DATA_BLOCK "BR04_TR07"	// DB 240
VERSION : 0.1
  STRUCT
   Front : STRUCT
    Hook : ARRAY  [1 .. 10 ] OF UDT 102;
   END_STRUCT ;
   Rear : STRUCT
    Hook : ARRAY  [1 .. 10 ] OF UDT 102;
   END_STRUCT ;
  END_STRUCT ;	
BEGIN
   Front.Hook[1].HookOver := L#6716;
   Front.Hook[1].HookUnderOffset := L#115;
   Front.Hook[1].TelPos_1.TelPos := L#3;
   Front.Hook[2].HookOver := L#5745;
   Front.Hook[2].HookUnderOffset := L#115;
   Front.Hook[2].TelPos_1.TelPos := L#3;
   Front.Hook[3].HookOver := L#4775;
   Front.Hook[3].HookUnderOffset := L#115;
   Front.Hook[3].TelPos_1.TelPos := L#3;
   Front.Hook[4].HookOver := L#3805;
   Front.Hook[4].HookUnderOffset := L#115;
   Front.Hook[4].TelPos_1.TelPos := L#3;
   Front.Hook[5].HookOver := L#2835;
   Front.Hook[5].HookUnderOffset := L#115;
   Front.Hook[5].TelPos_1.TelPos := L#3;
   Front.Hook[6].HookOver := L#1865;
   Front.Hook[6].HookUnderOffset := L#115;
   Front.Hook[6].TelPos_1.TelPos := L#3;
   Rear.Hook[1].HookOver := L#6716;
   Rear.Hook[1].HookUnderOffset := L#115;
   Rear.Hook[1].TelPos_1.TelPos := L#4;
   Rear.Hook[2].HookOver := L#5745;
   Rear.Hook[2].HookUnderOffset := L#115;
   Rear.Hook[2].TelPos_1.TelPos := L#4;
   Rear.Hook[3].HookOver := L#4775;
   Rear.Hook[3].HookUnderOffset := L#115;
   Rear.Hook[3].TelPos_1.TelPos := L#4;
   Rear.Hook[4].HookOver := L#3805;
   Rear.Hook[4].HookUnderOffset := L#115;
   Rear.Hook[4].TelPos_1.TelPos := L#4;
   Rear.Hook[5].HookOver := L#2835;
   Rear.Hook[5].HookUnderOffset := L#115;
   Rear.Hook[5].TelPos_1.TelPos := L#4;
   Rear.Hook[6].HookOver := L#1865;
   Rear.Hook[6].HookUnderOffset := L#115;
   Rear.Hook[6].TelPos_1.TelPos := L#4;
END_DATA_BLOCK

DATA_BLOCK "BR04_TR08"	// DB 241
VERSION : 0.1
  STRUCT
   Front : STRUCT
    Hook : ARRAY  [1 .. 10 ] OF UDT 102;
   END_STRUCT ;
   Rear : STRUCT
    Hook : ARRAY  [1 .. 10 ] OF UDT 102;
   END_STRUCT ;
  END_STRUCT ;	
BEGIN
   Front.Hook[1].HookOver := L#6716;
   Front.Hook[1].HookUnderOffset := L#115;
   Front.Hook[1].TelPos_1.TelPos := L#3;
   Front.Hook[2].HookOver := L#5745;
   Front.Hook[2].HookUnderOffset := L#115;
   Front.Hook[2].TelPos_1.TelPos := L#3;
   Front.Hook[3].HookOver := L#4775;
   Front.Hook[3].HookUnderOffset := L#115;
   Front.Hook[3].TelPos_1.TelPos := L#3;
   Front.Hook[4].HookOver := L#3805;
   Front.Hook[4].HookUnderOffset := L#115;
   Front.Hook[4].TelPos_1.TelPos := L#3;
   Front.Hook[5].HookOver := L#2835;
   Front.Hook[5].HookUnderOffset := L#115;
   Front.Hook[5].TelPos_1.TelPos := L#3;
   Front.Hook[6].HookOver := L#1865;
   Front.Hook[6].HookUnderOffset := L#115;
   Front.Hook[6].TelPos_1.TelPos := L#3;
   Rear.Hook[1].HookOver := L#6716;
   Rear.Hook[1].HookUnderOffset := L#115;
   Rear.Hook[1].TelPos_1.TelPos := L#4;
   Rear.Hook[2].HookOver := L#5745;
   Rear.Hook[2].HookUnderOffset := L#115;
   Rear.Hook[2].TelPos_1.TelPos := L#4;
   Rear.Hook[3].HookOver := L#4775;
   Rear.Hook[3].HookUnderOffset := L#115;
   Rear.Hook[3].TelPos_1.TelPos := L#4;
   Rear.Hook[4].HookOver := L#3805;
   Rear.Hook[4].HookUnderOffset := L#115;
   Rear.Hook[4].TelPos_1.TelPos := L#4;
   Rear.Hook[5].HookOver := L#2835;
   Rear.Hook[5].HookUnderOffset := L#115;
   Rear.Hook[5].TelPos_1.TelPos := L#4;
   Rear.Hook[6].HookOver := L#1865;
   Rear.Hook[6].HookUnderOffset := L#115;
   Rear.Hook[6].TelPos_1.TelPos := L#4;
END_DATA_BLOCK

DATA_BLOCK "BR04_TR09"	// DB 242
VERSION : 0.1
  STRUCT
   Front : STRUCT
    Hook : ARRAY  [1 .. 10 ] OF UDT 102;
   END_STRUCT ;
   Rear : STRUCT
    Hook : ARRAY  [1 .. 10 ] OF UDT 102;
   END_STRUCT ;
  END_STRUCT ;	
BEGIN
   Front.Hook[1].HookOver := L#6716;
   Front.Hook[1].HookUnderOffset := L#115;
   Front.Hook[1].TelPos_1.TelPos := L#3;
   Front.Hook[2].HookOver := L#5745;
   Front.Hook[2].HookUnderOffset := L#115;
   Front.Hook[2].TelPos_1.TelPos := L#3;
   Front.Hook[3].HookOver := L#4775;
   Front.Hook[3].HookUnderOffset := L#115;
   Front.Hook[3].TelPos_1.TelPos := L#3;
   Front.Hook[4].HookOver := L#3805;
   Front.Hook[4].HookUnderOffset := L#115;
   Front.Hook[4].TelPos_1.TelPos := L#3;
   Front.Hook[5].HookOver := L#2835;
   Front.Hook[5].HookUnderOffset := L#115;
   Front.Hook[5].TelPos_1.TelPos := L#3;
   Front.Hook[6].HookOver := L#1865;
   Front.Hook[6].HookUnderOffset := L#115;
   Front.Hook[6].TelPos_1.TelPos := L#3;
   Rear.Hook[1].HookOver := L#6716;
   Rear.Hook[1].HookUnderOffset := L#115;
   Rear.Hook[1].TelPos_1.TelPos := L#4;
   Rear.Hook[2].HookOver := L#5745;
   Rear.Hook[2].HookUnderOffset := L#115;
   Rear.Hook[2].TelPos_1.TelPos := L#4;
   Rear.Hook[3].HookOver := L#4775;
   Rear.Hook[3].HookUnderOffset := L#115;
   Rear.Hook[3].TelPos_1.TelPos := L#4;
   Rear.Hook[4].HookOver := L#3805;
   Rear.Hook[4].HookUnderOffset := L#115;
   Rear.Hook[4].TelPos_1.TelPos := L#4;
   Rear.Hook[5].HookOver := L#2835;
   Rear.Hook[5].HookUnderOffset := L#115;
   Rear.Hook[5].TelPos_1.TelPos := L#4;
   Rear.Hook[6].HookOver := L#1865;
   Rear.Hook[6].HookUnderOffset := L#115;
   Rear.Hook[6].TelPos_1.TelPos := L#4;
END_DATA_BLOCK

DATA_BLOCK "BR04_TR10"	// DB 243
VERSION : 0.1
  STRUCT
   Front : STRUCT
    Hook : ARRAY  [1 .. 10 ] OF UDT 102;
   END_STRUCT ;
   Rear : STRUCT
    Hook : ARRAY  [1 .. 10 ] OF UDT 102;
   END_STRUCT ;
  END_STRUCT ;	
BEGIN
   Front.Hook[1].HookOver := L#6716;
   Front.Hook[1].HookUnderOffset := L#115;
   Front.Hook[1].TelPos_1.TelPos := L#3;
   Front.Hook[2].HookOver := L#5745;
   Front.Hook[2].HookUnderOffset := L#115;
   Front.Hook[2].TelPos_1.TelPos := L#3;
   Front.Hook[3].HookOver := L#4775;
   Front.Hook[3].HookUnderOffset := L#115;
   Front.Hook[3].TelPos_1.TelPos := L#3;
   Front.Hook[4].HookOver := L#3805;
   Front.Hook[4].HookUnderOffset := L#115;
   Front.Hook[4].TelPos_1.TelPos := L#3;
   Front.Hook[5].HookOver := L#2835;
   Front.Hook[5].HookUnderOffset := L#115;
   Front.Hook[5].TelPos_1.TelPos := L#3;
   Rear.Hook[1].HookOver := L#6716;
   Rear.Hook[1].HookUnderOffset := L#115;
   Rear.Hook[1].TelPos_1.TelPos := L#4;
   Rear.Hook[2].HookOver := L#5745;
   Rear.Hook[2].HookUnderOffset := L#115;
   Rear.Hook[2].TelPos_1.TelPos := L#4;
   Rear.Hook[3].HookOver := L#4775;
   Rear.Hook[3].HookUnderOffset := L#115;
   Rear.Hook[3].TelPos_1.TelPos := L#4;
   Rear.Hook[4].HookOver := L#3805;
   Rear.Hook[4].HookUnderOffset := L#115;
   Rear.Hook[4].TelPos_1.TelPos := L#4;
   Rear.Hook[5].HookOver := L#2835;
   Rear.Hook[5].HookUnderOffset := L#115;
   Rear.Hook[5].TelPos_1.TelPos := L#4;
END_DATA_BLOCK

DATA_BLOCK "BR04_TR11"	// DB 244
VERSION : 0.1
  STRUCT
   Front : STRUCT
    Hook : ARRAY  [1 .. 10 ] OF UDT 102;
   END_STRUCT ;
   Rear : STRUCT
    Hook : ARRAY  [1 .. 10 ] OF UDT 102;
   END_STRUCT ;
  END_STRUCT ;	
BEGIN
   Front.Hook[1].HookOver := L#6716;
   Front.Hook[1].HookUnderOffset := L#115;
   Front.Hook[1].TelPos_1.TelPos := L#3;
   Front.Hook[2].HookOver := L#5745;
   Front.Hook[2].HookUnderOffset := L#115;
   Front.Hook[2].TelPos_1.TelPos := L#3;
   Front.Hook[3].HookOver := L#4775;
   Front.Hook[3].HookUnderOffset := L#115;
   Front.Hook[3].TelPos_1.TelPos := L#3;
   Front.Hook[4].HookOver := L#3805;
   Front.Hook[4].HookUnderOffset := L#115;
   Front.Hook[4].TelPos_1.TelPos := L#3;
   Front.Hook[5].HookOver := L#2835;
   Front.Hook[5].HookUnderOffset := L#115;
   Front.Hook[5].TelPos_1.TelPos := L#3;
   Front.Hook[6].HookOver := L#1865;
   Front.Hook[6].HookUnderOffset := L#115;
   Front.Hook[6].TelPos_1.TelPos := L#3;
   Rear.Hook[1].HookOver := L#6716;
   Rear.Hook[1].HookUnderOffset := L#115;
   Rear.Hook[1].TelPos_1.TelPos := L#4;
   Rear.Hook[2].HookOver := L#5745;
   Rear.Hook[2].HookUnderOffset := L#115;
   Rear.Hook[2].TelPos_1.TelPos := L#4;
   Rear.Hook[3].HookOver := L#4775;
   Rear.Hook[3].HookUnderOffset := L#115;
   Rear.Hook[3].TelPos_1.TelPos := L#4;
   Rear.Hook[4].HookOver := L#3805;
   Rear.Hook[4].HookUnderOffset := L#115;
   Rear.Hook[4].TelPos_1.TelPos := L#4;
   Rear.Hook[5].HookOver := L#2835;
   Rear.Hook[5].HookUnderOffset := L#115;
   Rear.Hook[5].TelPos_1.TelPos := L#4;
   Rear.Hook[6].HookOver := L#1865;
   Rear.Hook[6].HookUnderOffset := L#115;
   Rear.Hook[6].TelPos_1.TelPos := L#4;
END_DATA_BLOCK

DATA_BLOCK "BR05_TR01"	// DB 245
VERSION : 0.1
  STRUCT
   Front : STRUCT
    Hook : ARRAY  [1 .. 10 ] OF UDT 102;
   END_STRUCT ;
   Rear : STRUCT
    Hook : ARRAY  [1 .. 10 ] OF UDT 102;
   END_STRUCT ;
  END_STRUCT ;	
BEGIN
   Front.Hook[1].HookOver := L#6716;
   Front.Hook[1].HookUnderOffset := L#115;
   Front.Hook[1].TelPos_1.TelPos := L#3;
   Front.Hook[2].HookOver := L#5745;
   Front.Hook[2].HookUnderOffset := L#115;
   Front.Hook[2].TelPos_1.TelPos := L#3;
   Front.Hook[3].HookOver := L#4775;
   Front.Hook[3].HookUnderOffset := L#115;
   Front.Hook[3].TelPos_1.TelPos := L#3;
   Front.Hook[4].HookOver := L#3805;
   Front.Hook[4].HookUnderOffset := L#115;
   Front.Hook[4].TelPos_1.TelPos := L#3;
   Front.Hook[5].HookOver := L#2835;
   Front.Hook[5].HookUnderOffset := L#115;
   Front.Hook[5].TelPos_1.TelPos := L#3;
   Rear.Hook[1].HookOver := L#6716;
   Rear.Hook[1].HookUnderOffset := L#115;
   Rear.Hook[1].TelPos_1.TelPos := L#4;
   Rear.Hook[2].HookOver := L#5745;
   Rear.Hook[2].HookUnderOffset := L#115;
   Rear.Hook[2].TelPos_1.TelPos := L#4;
   Rear.Hook[3].HookOver := L#4775;
   Rear.Hook[3].HookUnderOffset := L#115;
   Rear.Hook[3].TelPos_1.TelPos := L#4;
   Rear.Hook[4].HookOver := L#3805;
   Rear.Hook[4].HookUnderOffset := L#115;
   Rear.Hook[4].TelPos_1.TelPos := L#4;
   Rear.Hook[5].HookOver := L#2835;
   Rear.Hook[5].HookUnderOffset := L#115;
   Rear.Hook[5].TelPos_1.TelPos := L#4;
END_DATA_BLOCK

DATA_BLOCK "BR05_TR02"	// DB 246
VERSION : 0.1
  STRUCT
   Front : STRUCT
    Hook : ARRAY  [1 .. 10 ] OF UDT 102;
   END_STRUCT ;
   Rear : STRUCT
    Hook : ARRAY  [1 .. 10 ] OF UDT 102;
   END_STRUCT ;
  END_STRUCT ;	
BEGIN
   Front.Hook[1].HookOver := L#6716;
   Front.Hook[1].HookUnderOffset := L#115;
   Front.Hook[1].TelPos_1.TelPos := L#3;
   Front.Hook[2].HookOver := L#5745;
   Front.Hook[2].HookUnderOffset := L#115;
   Front.Hook[2].TelPos_1.TelPos := L#3;
   Front.Hook[3].HookOver := L#4775;
   Front.Hook[3].HookUnderOffset := L#115;
   Front.Hook[3].TelPos_1.TelPos := L#3;
   Front.Hook[4].HookOver := L#3805;
   Front.Hook[4].HookUnderOffset := L#115;
   Front.Hook[4].TelPos_1.TelPos := L#3;
   Front.Hook[5].HookOver := L#2835;
   Front.Hook[5].HookUnderOffset := L#115;
   Front.Hook[5].TelPos_1.TelPos := L#3;
   Front.Hook[6].HookOver := L#1865;
   Front.Hook[6].HookUnderOffset := L#115;
   Front.Hook[6].TelPos_1.TelPos := L#3;
   Rear.Hook[1].HookOver := L#6716;
   Rear.Hook[1].HookUnderOffset := L#115;
   Rear.Hook[1].TelPos_1.TelPos := L#4;
   Rear.Hook[2].HookOver := L#5745;
   Rear.Hook[2].HookUnderOffset := L#115;
   Rear.Hook[2].TelPos_1.TelPos := L#4;
   Rear.Hook[3].HookOver := L#4775;
   Rear.Hook[3].HookUnderOffset := L#115;
   Rear.Hook[3].TelPos_1.TelPos := L#4;
   Rear.Hook[4].HookOver := L#3805;
   Rear.Hook[4].HookUnderOffset := L#115;
   Rear.Hook[4].TelPos_1.TelPos := L#4;
   Rear.Hook[5].HookOver := L#2835;
   Rear.Hook[5].HookUnderOffset := L#115;
   Rear.Hook[5].TelPos_1.TelPos := L#4;
   Rear.Hook[6].HookOver := L#1865;
   Rear.Hook[6].HookUnderOffset := L#115;
   Rear.Hook[6].TelPos_1.TelPos := L#4;
END_DATA_BLOCK

DATA_BLOCK "BR05_TR03"	// DB 247
VERSION : 0.1
  STRUCT
   Front : STRUCT
    Hook : ARRAY  [1 .. 10 ] OF UDT 102;
   END_STRUCT ;
   Rear : STRUCT
    Hook : ARRAY  [1 .. 10 ] OF UDT 102;
   END_STRUCT ;
  END_STRUCT ;	
BEGIN
   Front.Hook[1].HookOver := L#6716;
   Front.Hook[1].HookUnderOffset := L#115;
   Front.Hook[1].TelPos_1.TelPos := L#3;
   Front.Hook[2].HookOver := L#5745;
   Front.Hook[2].HookUnderOffset := L#115;
   Front.Hook[2].TelPos_1.TelPos := L#3;
   Front.Hook[3].HookOver := L#4775;
   Front.Hook[3].HookUnderOffset := L#115;
   Front.Hook[3].TelPos_1.TelPos := L#3;
   Front.Hook[4].HookOver := L#3805;
   Front.Hook[4].HookUnderOffset := L#115;
   Front.Hook[4].TelPos_1.TelPos := L#3;
   Front.Hook[5].HookOver := L#2835;
   Front.Hook[5].HookUnderOffset := L#115;
   Front.Hook[5].TelPos_1.TelPos := L#3;
   Front.Hook[6].HookOver := L#1865;
   Front.Hook[6].HookUnderOffset := L#115;
   Front.Hook[6].TelPos_1.TelPos := L#3;
   Rear.Hook[1].HookOver := L#6716;
   Rear.Hook[1].HookUnderOffset := L#115;
   Rear.Hook[1].TelPos_1.TelPos := L#4;
   Rear.Hook[2].HookOver := L#5745;
   Rear.Hook[2].HookUnderOffset := L#115;
   Rear.Hook[2].TelPos_1.TelPos := L#4;
   Rear.Hook[3].HookOver := L#4775;
   Rear.Hook[3].HookUnderOffset := L#115;
   Rear.Hook[3].TelPos_1.TelPos := L#4;
   Rear.Hook[4].HookOver := L#3805;
   Rear.Hook[4].HookUnderOffset := L#115;
   Rear.Hook[4].TelPos_1.TelPos := L#4;
   Rear.Hook[5].HookOver := L#2835;
   Rear.Hook[5].HookUnderOffset := L#115;
   Rear.Hook[5].TelPos_1.TelPos := L#4;
   Rear.Hook[6].HookOver := L#1865;
   Rear.Hook[6].HookUnderOffset := L#115;
   Rear.Hook[6].TelPos_1.TelPos := L#4;
END_DATA_BLOCK

DATA_BLOCK "BR05_TR04"	// DB 248
VERSION : 0.1
  STRUCT
   Front : STRUCT
    Hook : ARRAY  [1 .. 10 ] OF UDT 102;
   END_STRUCT ;
   Rear : STRUCT
    Hook : ARRAY  [1 .. 10 ] OF UDT 102;
   END_STRUCT ;
  END_STRUCT ;	
BEGIN
   Front.Hook[1].HookOver := L#6716;
   Front.Hook[1].HookUnderOffset := L#115;
   Front.Hook[1].TelPos_1.TelPos := L#3;
   Front.Hook[2].HookOver := L#5745;
   Front.Hook[2].HookUnderOffset := L#115;
   Front.Hook[2].TelPos_1.TelPos := L#3;
   Front.Hook[3].HookOver := L#4775;
   Front.Hook[3].HookUnderOffset := L#115;
   Front.Hook[3].TelPos_1.TelPos := L#3;
   Front.Hook[4].HookOver := L#3805;
   Front.Hook[4].HookUnderOffset := L#115;
   Front.Hook[4].TelPos_1.TelPos := L#3;
   Front.Hook[5].HookOver := L#2835;
   Front.Hook[5].HookUnderOffset := L#115;
   Front.Hook[5].TelPos_1.TelPos := L#3;
   Front.Hook[6].HookOver := L#1865;
   Front.Hook[6].HookUnderOffset := L#115;
   Front.Hook[6].TelPos_1.TelPos := L#3;
   Rear.Hook[1].HookOver := L#6716;
   Rear.Hook[1].HookUnderOffset := L#115;
   Rear.Hook[1].TelPos_1.TelPos := L#4;
   Rear.Hook[2].HookOver := L#5745;
   Rear.Hook[2].HookUnderOffset := L#115;
   Rear.Hook[2].TelPos_1.TelPos := L#4;
   Rear.Hook[3].HookOver := L#4775;
   Rear.Hook[3].HookUnderOffset := L#115;
   Rear.Hook[3].TelPos_1.TelPos := L#4;
   Rear.Hook[4].HookOver := L#3805;
   Rear.Hook[4].HookUnderOffset := L#115;
   Rear.Hook[4].TelPos_1.TelPos := L#4;
   Rear.Hook[5].HookOver := L#2835;
   Rear.Hook[5].HookUnderOffset := L#115;
   Rear.Hook[5].TelPos_1.TelPos := L#4;
   Rear.Hook[6].HookOver := L#1865;
   Rear.Hook[6].HookUnderOffset := L#115;
   Rear.Hook[6].TelPos_1.TelPos := L#4;
END_DATA_BLOCK

DATA_BLOCK "BR05_TR05"	// DB 249
VERSION : 0.1
  STRUCT
   Front : STRUCT
    Hook : ARRAY  [1 .. 10 ] OF UDT 102;
   END_STRUCT ;
   Rear : STRUCT
    Hook : ARRAY  [1 .. 10 ] OF UDT 102;
   END_STRUCT ;
  END_STRUCT ;	
BEGIN
   Front.Hook[1].HookOver := L#6716;
   Front.Hook[1].HookUnderOffset := L#115;
   Front.Hook[1].TelPos_1.TelPos := L#3;
   Front.Hook[2].HookOver := L#5745;
   Front.Hook[2].HookUnderOffset := L#115;
   Front.Hook[2].TelPos_1.TelPos := L#3;
   Front.Hook[3].HookOver := L#4775;
   Front.Hook[3].HookUnderOffset := L#115;
   Front.Hook[3].TelPos_1.TelPos := L#3;
   Front.Hook[4].HookOver := L#3805;
   Front.Hook[4].HookUnderOffset := L#115;
   Front.Hook[4].TelPos_1.TelPos := L#3;
   Front.Hook[5].HookOver := L#2835;
   Front.Hook[5].HookUnderOffset := L#115;
   Front.Hook[5].TelPos_1.TelPos := L#3;
   Front.Hook[6].HookOver := L#1865;
   Front.Hook[6].HookUnderOffset := L#115;
   Front.Hook[6].TelPos_1.TelPos := L#3;
   Rear.Hook[1].HookOver := L#6716;
   Rear.Hook[1].HookUnderOffset := L#115;
   Rear.Hook[1].TelPos_1.TelPos := L#4;
   Rear.Hook[2].HookOver := L#5745;
   Rear.Hook[2].HookUnderOffset := L#115;
   Rear.Hook[2].TelPos_1.TelPos := L#4;
   Rear.Hook[3].HookOver := L#4775;
   Rear.Hook[3].HookUnderOffset := L#115;
   Rear.Hook[3].TelPos_1.TelPos := L#4;
   Rear.Hook[4].HookOver := L#3805;
   Rear.Hook[4].HookUnderOffset := L#115;
   Rear.Hook[4].TelPos_1.TelPos := L#4;
   Rear.Hook[5].HookOver := L#2835;
   Rear.Hook[5].HookUnderOffset := L#115;
   Rear.Hook[5].TelPos_1.TelPos := L#4;
   Rear.Hook[6].HookOver := L#1865;
   Rear.Hook[6].HookUnderOffset := L#115;
   Rear.Hook[6].TelPos_1.TelPos := L#4;
END_DATA_BLOCK

DATA_BLOCK "BR05_TR06"	// DB 250
VERSION : 0.1
  STRUCT
   Front : STRUCT
    Hook : ARRAY  [1 .. 10 ] OF UDT 102;
   END_STRUCT ;
   Rear : STRUCT
    Hook : ARRAY  [1 .. 10 ] OF UDT 102;
   END_STRUCT ;
  END_STRUCT ;	
BEGIN
   Front.Hook[1].HookOver := L#6716;
   Front.Hook[1].HookUnderOffset := L#115;
   Front.Hook[1].TelPos_1.TelPos := L#3;
   Front.Hook[2].HookOver := L#5745;
   Front.Hook[2].HookUnderOffset := L#115;
   Front.Hook[2].TelPos_1.TelPos := L#3;
   Front.Hook[3].HookOver := L#4775;
   Front.Hook[3].HookUnderOffset := L#115;
   Front.Hook[3].TelPos_1.TelPos := L#3;
   Front.Hook[4].HookOver := L#3805;
   Front.Hook[4].HookUnderOffset := L#115;
   Front.Hook[4].TelPos_1.TelPos := L#3;
   Front.Hook[5].HookOver := L#2835;
   Front.Hook[5].HookUnderOffset := L#115;
   Front.Hook[5].TelPos_1.TelPos := L#3;
   Front.Hook[6].HookOver := L#1865;
   Front.Hook[6].HookUnderOffset := L#115;
   Front.Hook[6].TelPos_1.TelPos := L#3;
   Rear.Hook[1].HookOver := L#6716;
   Rear.Hook[1].HookUnderOffset := L#115;
   Rear.Hook[1].TelPos_1.TelPos := L#4;
   Rear.Hook[2].HookOver := L#5745;
   Rear.Hook[2].HookUnderOffset := L#115;
   Rear.Hook[2].TelPos_1.TelPos := L#4;
   Rear.Hook[3].HookOver := L#4775;
   Rear.Hook[3].HookUnderOffset := L#115;
   Rear.Hook[3].TelPos_1.TelPos := L#4;
   Rear.Hook[4].HookOver := L#3805;
   Rear.Hook[4].HookUnderOffset := L#115;
   Rear.Hook[4].TelPos_1.TelPos := L#4;
   Rear.Hook[5].HookOver := L#2835;
   Rear.Hook[5].HookUnderOffset := L#115;
   Rear.Hook[5].TelPos_1.TelPos := L#4;
   Rear.Hook[6].HookOver := L#1865;
   Rear.Hook[6].HookUnderOffset := L#115;
   Rear.Hook[6].TelPos_1.TelPos := L#4;
END_DATA_BLOCK

DATA_BLOCK "BR05_TR07"	// DB 251
VERSION : 0.1
  STRUCT
   Front : STRUCT
    Hook : ARRAY  [1 .. 10 ] OF UDT 102;
   END_STRUCT ;
   Rear : STRUCT
    Hook : ARRAY  [1 .. 10 ] OF UDT 102;
   END_STRUCT ;
  END_STRUCT ;	
BEGIN
   Front.Hook[1].HookOver := L#6716;
   Front.Hook[1].HookUnderOffset := L#115;
   Front.Hook[1].TelPos_1.TelPos := L#3;
   Front.Hook[2].HookOver := L#5745;
   Front.Hook[2].HookUnderOffset := L#115;
   Front.Hook[2].TelPos_1.TelPos := L#3;
   Front.Hook[3].HookOver := L#4775;
   Front.Hook[3].HookUnderOffset := L#115;
   Front.Hook[3].TelPos_1.TelPos := L#3;
   Front.Hook[4].HookOver := L#3805;
   Front.Hook[4].HookUnderOffset := L#115;
   Front.Hook[4].TelPos_1.TelPos := L#3;
   Front.Hook[5].HookOver := L#2835;
   Front.Hook[5].HookUnderOffset := L#115;
   Front.Hook[5].TelPos_1.TelPos := L#3;
   Front.Hook[6].HookOver := L#1865;
   Front.Hook[6].HookUnderOffset := L#115;
   Front.Hook[6].TelPos_1.TelPos := L#3;
   Rear.Hook[1].HookOver := L#6716;
   Rear.Hook[1].HookUnderOffset := L#115;
   Rear.Hook[1].TelPos_1.TelPos := L#4;
   Rear.Hook[2].HookOver := L#5745;
   Rear.Hook[2].HookUnderOffset := L#115;
   Rear.Hook[2].TelPos_1.TelPos := L#4;
   Rear.Hook[3].HookOver := L#4775;
   Rear.Hook[3].HookUnderOffset := L#115;
   Rear.Hook[3].TelPos_1.TelPos := L#4;
   Rear.Hook[4].HookOver := L#3805;
   Rear.Hook[4].HookUnderOffset := L#115;
   Rear.Hook[4].TelPos_1.TelPos := L#4;
   Rear.Hook[5].HookOver := L#2835;
   Rear.Hook[5].HookUnderOffset := L#115;
   Rear.Hook[5].TelPos_1.TelPos := L#4;
   Rear.Hook[6].HookOver := L#1865;
   Rear.Hook[6].HookUnderOffset := L#115;
   Rear.Hook[6].TelPos_1.TelPos := L#4;
END_DATA_BLOCK

DATA_BLOCK "BR05_TR08"	// DB 252
VERSION : 0.1
  STRUCT
   Front : STRUCT
    Hook : ARRAY  [1 .. 10 ] OF UDT 102;
   END_STRUCT ;
   Rear : STRUCT
    Hook : ARRAY  [1 .. 10 ] OF UDT 102;
   END_STRUCT ;
  END_STRUCT ;	
BEGIN
   Front.Hook[1].HookOver := L#6716;
   Front.Hook[1].HookUnderOffset := L#115;
   Front.Hook[1].TelPos_1.TelPos := L#3;
   Front.Hook[2].HookOver := L#5745;
   Front.Hook[2].HookUnderOffset := L#115;
   Front.Hook[2].TelPos_1.TelPos := L#3;
   Front.Hook[3].HookOver := L#4775;
   Front.Hook[3].HookUnderOffset := L#115;
   Front.Hook[3].TelPos_1.TelPos := L#3;
   Front.Hook[4].HookOver := L#3805;
   Front.Hook[4].HookUnderOffset := L#115;
   Front.Hook[4].TelPos_1.TelPos := L#3;
   Front.Hook[5].HookOver := L#2835;
   Front.Hook[5].HookUnderOffset := L#115;
   Front.Hook[5].TelPos_1.TelPos := L#3;
   Front.Hook[6].HookOver := L#1865;
   Front.Hook[6].HookUnderOffset := L#115;
   Front.Hook[6].TelPos_1.TelPos := L#3;
   Rear.Hook[1].HookOver := L#6716;
   Rear.Hook[1].HookUnderOffset := L#115;
   Rear.Hook[1].TelPos_1.TelPos := L#4;
   Rear.Hook[2].HookOver := L#5745;
   Rear.Hook[2].HookUnderOffset := L#115;
   Rear.Hook[2].TelPos_1.TelPos := L#4;
   Rear.Hook[3].HookOver := L#4775;
   Rear.Hook[3].HookUnderOffset := L#115;
   Rear.Hook[3].TelPos_1.TelPos := L#4;
   Rear.Hook[4].HookOver := L#3805;
   Rear.Hook[4].HookUnderOffset := L#115;
   Rear.Hook[4].TelPos_1.TelPos := L#4;
   Rear.Hook[5].HookOver := L#2835;
   Rear.Hook[5].HookUnderOffset := L#115;
   Rear.Hook[5].TelPos_1.TelPos := L#4;
   Rear.Hook[6].HookOver := L#1865;
   Rear.Hook[6].HookUnderOffset := L#115;
   Rear.Hook[6].TelPos_1.TelPos := L#4;
END_DATA_BLOCK

DATA_BLOCK "BR05_TR09"	// DB 253
VERSION : 0.1
  STRUCT
   Front : STRUCT
    Hook : ARRAY  [1 .. 10 ] OF UDT 102;
   END_STRUCT ;
   Rear : STRUCT
    Hook : ARRAY  [1 .. 10 ] OF UDT 102;
   END_STRUCT ;
  END_STRUCT ;	
BEGIN
   Front.Hook[1].HookOver := L#6716;
   Front.Hook[1].HookUnderOffset := L#115;
   Front.Hook[1].TelPos_1.TelPos := L#3;
   Front.Hook[2].HookOver := L#5745;
   Front.Hook[2].HookUnderOffset := L#115;
   Front.Hook[2].TelPos_1.TelPos := L#3;
   Front.Hook[3].HookOver := L#4775;
   Front.Hook[3].HookUnderOffset := L#115;
   Front.Hook[3].TelPos_1.TelPos := L#3;
   Front.Hook[4].HookOver := L#3805;
   Front.Hook[4].HookUnderOffset := L#115;
   Front.Hook[4].TelPos_1.TelPos := L#3;
   Front.Hook[5].HookOver := L#2835;
   Front.Hook[5].HookUnderOffset := L#115;
   Front.Hook[5].TelPos_1.TelPos := L#3;
   Front.Hook[6].HookOver := L#1865;
   Front.Hook[6].HookUnderOffset := L#115;
   Front.Hook[6].TelPos_1.TelPos := L#3;
   Rear.Hook[1].HookOver := L#6716;
   Rear.Hook[1].HookUnderOffset := L#115;
   Rear.Hook[1].TelPos_1.TelPos := L#4;
   Rear.Hook[2].HookOver := L#5745;
   Rear.Hook[2].HookUnderOffset := L#115;
   Rear.Hook[2].TelPos_1.TelPos := L#4;
   Rear.Hook[3].HookOver := L#4775;
   Rear.Hook[3].HookUnderOffset := L#115;
   Rear.Hook[3].TelPos_1.TelPos := L#4;
   Rear.Hook[4].HookOver := L#3805;
   Rear.Hook[4].HookUnderOffset := L#115;
   Rear.Hook[4].TelPos_1.TelPos := L#4;
   Rear.Hook[5].HookOver := L#2835;
   Rear.Hook[5].HookUnderOffset := L#115;
   Rear.Hook[5].TelPos_1.TelPos := L#4;
   Rear.Hook[6].HookOver := L#1865;
   Rear.Hook[6].HookUnderOffset := L#115;
   Rear.Hook[6].TelPos_1.TelPos := L#4;
END_DATA_BLOCK

DATA_BLOCK "BR05_TR10"	// DB 254
VERSION : 0.1
  STRUCT
   Front : STRUCT
    Hook : ARRAY  [1 .. 10 ] OF UDT 102;
   END_STRUCT ;
   Rear : STRUCT
    Hook : ARRAY  [1 .. 10 ] OF UDT 102;
   END_STRUCT ;
  END_STRUCT ;	
BEGIN
   Front.Hook[1].HookOver := L#6716;
   Front.Hook[1].HookUnderOffset := L#115;
   Front.Hook[1].TelPos_1.TelPos := L#3;
   Front.Hook[2].HookOver := L#5745;
   Front.Hook[2].HookUnderOffset := L#115;
   Front.Hook[2].TelPos_1.TelPos := L#3;
   Front.Hook[3].HookOver := L#4775;
   Front.Hook[3].HookUnderOffset := L#115;
   Front.Hook[3].TelPos_1.TelPos := L#3;
   Front.Hook[4].HookOver := L#3805;
   Front.Hook[4].HookUnderOffset := L#115;
   Front.Hook[4].TelPos_1.TelPos := L#3;
   Front.Hook[5].HookOver := L#2835;
   Front.Hook[5].HookUnderOffset := L#115;
   Front.Hook[5].TelPos_1.TelPos := L#3;
   Rear.Hook[1].HookOver := L#6716;
   Rear.Hook[1].HookUnderOffset := L#115;
   Rear.Hook[1].TelPos_1.TelPos := L#4;
   Rear.Hook[2].HookOver := L#5745;
   Rear.Hook[2].HookUnderOffset := L#115;
   Rear.Hook[2].TelPos_1.TelPos := L#4;
   Rear.Hook[3].HookOver := L#4775;
   Rear.Hook[3].HookUnderOffset := L#115;
   Rear.Hook[3].TelPos_1.TelPos := L#4;
   Rear.Hook[4].HookOver := L#3805;
   Rear.Hook[4].HookUnderOffset := L#115;
   Rear.Hook[4].TelPos_1.TelPos := L#4;
   Rear.Hook[5].HookOver := L#2835;
   Rear.Hook[5].HookUnderOffset := L#115;
   Rear.Hook[5].TelPos_1.TelPos := L#4;
END_DATA_BLOCK

DATA_BLOCK "BR05_TR11"	// DB 255
VERSION : 0.1
  STRUCT
   Front : STRUCT
    Hook : ARRAY  [1 .. 10 ] OF UDT 102;
   END_STRUCT ;
   Rear : STRUCT
    Hook : ARRAY  [1 .. 10 ] OF UDT 102;
   END_STRUCT ;
  END_STRUCT ;	
BEGIN
   Front.Hook[1].HookOver := L#6716;
   Front.Hook[1].HookUnderOffset := L#115;
   Front.Hook[1].TelPos_1.TelPos := L#3;
   Front.Hook[2].HookOver := L#5745;
   Front.Hook[2].HookUnderOffset := L#115;
   Front.Hook[2].TelPos_1.TelPos := L#3;
   Front.Hook[3].HookOver := L#4775;
   Front.Hook[3].HookUnderOffset := L#115;
   Front.Hook[3].TelPos_1.TelPos := L#3;
   Front.Hook[4].HookOver := L#3805;
   Front.Hook[4].HookUnderOffset := L#115;
   Front.Hook[4].TelPos_1.TelPos := L#3;
   Front.Hook[5].HookOver := L#2835;
   Front.Hook[5].HookUnderOffset := L#115;
   Front.Hook[5].TelPos_1.TelPos := L#3;
   Front.Hook[6].HookOver := L#1865;
   Front.Hook[6].HookUnderOffset := L#115;
   Front.Hook[6].TelPos_1.TelPos := L#3;
   Rear.Hook[1].HookOver := L#6716;
   Rear.Hook[1].HookUnderOffset := L#115;
   Rear.Hook[1].TelPos_1.TelPos := L#4;
   Rear.Hook[2].HookOver := L#5745;
   Rear.Hook[2].HookUnderOffset := L#115;
   Rear.Hook[2].TelPos_1.TelPos := L#4;
   Rear.Hook[3].HookOver := L#4775;
   Rear.Hook[3].HookUnderOffset := L#115;
   Rear.Hook[3].TelPos_1.TelPos := L#4;
   Rear.Hook[4].HookOver := L#3805;
   Rear.Hook[4].HookUnderOffset := L#115;
   Rear.Hook[4].TelPos_1.TelPos := L#4;
   Rear.Hook[5].HookOver := L#2835;
   Rear.Hook[5].HookUnderOffset := L#115;
   Rear.Hook[5].TelPos_1.TelPos := L#4;
   Rear.Hook[6].HookOver := L#1865;
   Rear.Hook[6].HookUnderOffset := L#115;
   Rear.Hook[6].TelPos_1.TelPos := L#4;
END_DATA_BLOCK

DATA_BLOCK "BR06_TR01"	// DB 256
VERSION : 0.1
  STRUCT
   Front : STRUCT
    Hook : ARRAY  [1 .. 10 ] OF UDT 102;
   END_STRUCT ;
   Rear : STRUCT
    Hook : ARRAY  [1 .. 10 ] OF UDT 102;
   END_STRUCT ;
  END_STRUCT ;	
BEGIN
   Front.Hook[1].HookOver := L#6650;
   Front.Hook[1].HookUnderOffset := L#115;
   Front.Hook[1].TelPos_1.TelPos := L#1;
   Front.Hook[2].HookOver := L#5566;
   Front.Hook[2].HookUnderOffset := L#115;
   Front.Hook[2].TelPos_1.TelPos := L#1;
   Front.Hook[3].HookOver := L#4416;
   Front.Hook[3].HookUnderOffset := L#115;
   Front.Hook[3].TelPos_1.TelPos := L#1;
   Front.Hook[4].HookOver := L#3266;
   Front.Hook[4].HookUnderOffset := L#115;
   Front.Hook[4].TelPos_1.TelPos := L#1;
   Rear.Hook[1].HookOver := L#6716;
   Rear.Hook[1].HookUnderOffset := L#115;
   Rear.Hook[1].TelPos_1.TelPos := L#2;
   Rear.Hook[2].HookOver := L#5566;
   Rear.Hook[2].HookUnderOffset := L#115;
   Rear.Hook[2].TelPos_1.TelPos := L#2;
   Rear.Hook[3].HookOver := L#4416;
   Rear.Hook[3].HookUnderOffset := L#115;
   Rear.Hook[3].TelPos_1.TelPos := L#2;
   Rear.Hook[4].HookOver := L#3266;
   Rear.Hook[4].HookUnderOffset := L#115;
   Rear.Hook[4].TelPos_1.TelPos := L#2;
END_DATA_BLOCK

DATA_BLOCK "BR06_TR02"	// DB 257
VERSION : 0.1
  STRUCT
   Front : STRUCT
    Hook : ARRAY  [1 .. 10 ] OF UDT 102;
   END_STRUCT ;
   Rear : STRUCT
    Hook : ARRAY  [1 .. 10 ] OF UDT 102;
   END_STRUCT ;
  END_STRUCT ;	
BEGIN
   Front.Hook[1].HookOver := L#6703;
   Front.Hook[1].HookUnderOffset := L#115;
   Front.Hook[1].TelPos_1.TelPos := L#1;
   Front.Hook[2].HookOver := L#5560;
   Front.Hook[2].HookUnderOffset := L#115;
   Front.Hook[2].TelPos_1.TelPos := L#1;
   Front.Hook[3].HookOver := L#4415;
   Front.Hook[3].HookUnderOffset := L#115;
   Front.Hook[3].TelPos_1.TelPos := L#1;
   Front.Hook[4].HookOver := L#3260;
   Front.Hook[4].HookUnderOffset := L#115;
   Front.Hook[4].TelPos_1.TelPos := L#1;
   Front.Hook[5].HookOver := L#2115;
   Front.Hook[5].HookUnderOffset := L#115;
   Front.Hook[5].TelPos_1.TelPos := L#1;
   Rear.Hook[1].HookOver := L#6703;
   Rear.Hook[1].HookUnderOffset := L#115;
   Rear.Hook[1].TelPos_1.TelPos := L#2;
   Rear.Hook[2].HookOver := L#5560;
   Rear.Hook[2].HookUnderOffset := L#115;
   Rear.Hook[2].TelPos_1.TelPos := L#2;
   Rear.Hook[3].HookOver := L#4415;
   Rear.Hook[3].HookUnderOffset := L#115;
   Rear.Hook[3].TelPos_1.TelPos := L#2;
   Rear.Hook[4].HookOver := L#3260;
   Rear.Hook[4].HookUnderOffset := L#115;
   Rear.Hook[4].TelPos_1.TelPos := L#2;
   Rear.Hook[5].HookOver := L#2115;
   Rear.Hook[5].HookUnderOffset := L#115;
   Rear.Hook[5].TelPos_1.TelPos := L#2;
END_DATA_BLOCK

DATA_BLOCK "BR06_TR03"	// DB 258
VERSION : 0.1
  STRUCT
   Front : STRUCT
    Hook : ARRAY  [1 .. 10 ] OF UDT 102;
   END_STRUCT ;
   Rear : STRUCT
    Hook : ARRAY  [1 .. 10 ] OF UDT 102;
   END_STRUCT ;
  END_STRUCT ;	
BEGIN
   Front.Hook[1].HookOver := L#6703;
   Front.Hook[1].HookUnderOffset := L#115;
   Front.Hook[1].TelPos_1.TelPos := L#1;
   Front.Hook[2].HookOver := L#5560;
   Front.Hook[2].HookUnderOffset := L#115;
   Front.Hook[2].TelPos_1.TelPos := L#1;
   Front.Hook[3].HookOver := L#4415;
   Front.Hook[3].HookUnderOffset := L#115;
   Front.Hook[3].TelPos_1.TelPos := L#1;
   Front.Hook[4].HookOver := L#3260;
   Front.Hook[4].HookUnderOffset := L#115;
   Front.Hook[4].TelPos_1.TelPos := L#1;
   Front.Hook[5].HookOver := L#2115;
   Front.Hook[5].HookUnderOffset := L#115;
   Front.Hook[5].TelPos_1.TelPos := L#1;
   Rear.Hook[1].HookOver := L#6703;
   Rear.Hook[1].HookUnderOffset := L#115;
   Rear.Hook[1].TelPos_1.TelPos := L#2;
   Rear.Hook[2].HookOver := L#5560;
   Rear.Hook[2].HookUnderOffset := L#115;
   Rear.Hook[2].TelPos_1.TelPos := L#2;
   Rear.Hook[3].HookOver := L#4415;
   Rear.Hook[3].HookUnderOffset := L#115;
   Rear.Hook[3].TelPos_1.TelPos := L#2;
   Rear.Hook[4].HookOver := L#3260;
   Rear.Hook[4].HookUnderOffset := L#115;
   Rear.Hook[4].TelPos_1.TelPos := L#2;
   Rear.Hook[5].HookOver := L#2115;
   Rear.Hook[5].HookUnderOffset := L#115;
   Rear.Hook[5].TelPos_1.TelPos := L#2;
END_DATA_BLOCK

DATA_BLOCK "BR06_TR04"	// DB 259
VERSION : 0.1
  STRUCT
   Front : STRUCT
    Hook : ARRAY  [1 .. 10 ] OF UDT 102;
   END_STRUCT ;
   Rear : STRUCT
    Hook : ARRAY  [1 .. 10 ] OF UDT 102;
   END_STRUCT ;
  END_STRUCT ;	
BEGIN
   Front.Hook[1].HookOver := L#6703;
   Front.Hook[1].HookUnderOffset := L#115;
   Front.Hook[1].TelPos_1.TelPos := L#1;
   Front.Hook[2].HookOver := L#5560;
   Front.Hook[2].HookUnderOffset := L#115;
   Front.Hook[2].TelPos_1.TelPos := L#1;
   Front.Hook[3].HookOver := L#4415;
   Front.Hook[3].HookUnderOffset := L#115;
   Front.Hook[3].TelPos_1.TelPos := L#1;
   Front.Hook[4].HookOver := L#3260;
   Front.Hook[4].HookUnderOffset := L#115;
   Front.Hook[4].TelPos_1.TelPos := L#1;
   Front.Hook[5].HookOver := L#2115;
   Front.Hook[5].HookUnderOffset := L#115;
   Front.Hook[5].TelPos_1.TelPos := L#1;
   Rear.Hook[1].HookOver := L#6703;
   Rear.Hook[1].HookUnderOffset := L#115;
   Rear.Hook[1].TelPos_1.TelPos := L#2;
   Rear.Hook[2].HookOver := L#5560;
   Rear.Hook[2].HookUnderOffset := L#115;
   Rear.Hook[2].TelPos_1.TelPos := L#2;
   Rear.Hook[3].HookOver := L#4415;
   Rear.Hook[3].HookUnderOffset := L#115;
   Rear.Hook[3].TelPos_1.TelPos := L#2;
   Rear.Hook[4].HookOver := L#3260;
   Rear.Hook[4].HookUnderOffset := L#115;
   Rear.Hook[4].TelPos_1.TelPos := L#2;
   Rear.Hook[5].HookOver := L#2115;
   Rear.Hook[5].HookUnderOffset := L#115;
   Rear.Hook[5].TelPos_1.TelPos := L#2;
END_DATA_BLOCK

DATA_BLOCK "BR06_TR05"	// DB 260
VERSION : 0.1
  STRUCT
   Front : STRUCT
    Hook : ARRAY  [1 .. 10 ] OF UDT 102;
   END_STRUCT ;
   Rear : STRUCT
    Hook : ARRAY  [1 .. 10 ] OF UDT 102;
   END_STRUCT ;
  END_STRUCT ;	
BEGIN
   Front.Hook[1].HookOver := L#6703;
   Front.Hook[1].HookUnderOffset := L#115;
   Front.Hook[1].TelPos_1.TelPos := L#1;
   Front.Hook[2].HookOver := L#5560;
   Front.Hook[2].HookUnderOffset := L#115;
   Front.Hook[2].TelPos_1.TelPos := L#1;
   Front.Hook[3].HookOver := L#4415;
   Front.Hook[3].HookUnderOffset := L#115;
   Front.Hook[3].TelPos_1.TelPos := L#1;
   Front.Hook[4].HookOver := L#3260;
   Front.Hook[4].HookUnderOffset := L#115;
   Front.Hook[4].TelPos_1.TelPos := L#1;
   Front.Hook[5].HookOver := L#2115;
   Front.Hook[5].HookUnderOffset := L#115;
   Front.Hook[5].TelPos_1.TelPos := L#1;
   Rear.Hook[1].HookOver := L#6703;
   Rear.Hook[1].HookUnderOffset := L#115;
   Rear.Hook[1].TelPos_1.TelPos := L#2;
   Rear.Hook[2].HookOver := L#5560;
   Rear.Hook[2].HookUnderOffset := L#115;
   Rear.Hook[2].TelPos_1.TelPos := L#2;
   Rear.Hook[3].HookOver := L#4415;
   Rear.Hook[3].HookUnderOffset := L#115;
   Rear.Hook[3].TelPos_1.TelPos := L#2;
   Rear.Hook[4].HookOver := L#3260;
   Rear.Hook[4].HookUnderOffset := L#115;
   Rear.Hook[4].TelPos_1.TelPos := L#2;
   Rear.Hook[5].HookOver := L#2115;
   Rear.Hook[5].HookUnderOffset := L#115;
   Rear.Hook[5].TelPos_1.TelPos := L#2;
END_DATA_BLOCK

DATA_BLOCK "BR06_TR06"	// DB 261
VERSION : 0.1
  STRUCT
   Front : STRUCT
    Hook : ARRAY  [1 .. 10 ] OF UDT 102;
   END_STRUCT ;
   Rear : STRUCT
    Hook : ARRAY  [1 .. 10 ] OF UDT 102;
   END_STRUCT ;
  END_STRUCT ;	
BEGIN
   Front.Hook[1].HookOver := L#6703;
   Front.Hook[1].HookUnderOffset := L#115;
   Front.Hook[1].TelPos_1.TelPos := L#1;
   Front.Hook[2].HookOver := L#5560;
   Front.Hook[2].HookUnderOffset := L#115;
   Front.Hook[2].TelPos_1.TelPos := L#1;
   Front.Hook[3].HookOver := L#4415;
   Front.Hook[3].HookUnderOffset := L#115;
   Front.Hook[3].TelPos_1.TelPos := L#1;
   Front.Hook[4].HookOver := L#3260;
   Front.Hook[4].HookUnderOffset := L#115;
   Front.Hook[4].TelPos_1.TelPos := L#1;
   Front.Hook[5].HookOver := L#2115;
   Front.Hook[5].HookUnderOffset := L#115;
   Front.Hook[5].TelPos_1.TelPos := L#1;
   Rear.Hook[1].HookOver := L#6703;
   Rear.Hook[1].HookUnderOffset := L#115;
   Rear.Hook[1].TelPos_1.TelPos := L#2;
   Rear.Hook[2].HookOver := L#5560;
   Rear.Hook[2].HookUnderOffset := L#115;
   Rear.Hook[2].TelPos_1.TelPos := L#2;
   Rear.Hook[3].HookOver := L#4415;
   Rear.Hook[3].HookUnderOffset := L#115;
   Rear.Hook[3].TelPos_1.TelPos := L#2;
   Rear.Hook[4].HookOver := L#3260;
   Rear.Hook[4].HookUnderOffset := L#115;
   Rear.Hook[4].TelPos_1.TelPos := L#2;
   Rear.Hook[5].HookOver := L#2115;
   Rear.Hook[5].HookUnderOffset := L#115;
   Rear.Hook[5].TelPos_1.TelPos := L#2;
END_DATA_BLOCK

DATA_BLOCK "BR06_TR07"	// DB 262
VERSION : 0.1
  STRUCT
   Front : STRUCT
    Hook : ARRAY  [1 .. 10 ] OF UDT 102;
   END_STRUCT ;
   Rear : STRUCT
    Hook : ARRAY  [1 .. 10 ] OF UDT 102;
   END_STRUCT ;
  END_STRUCT ;	
BEGIN
   Front.Hook[1].HookOver := L#6703;
   Front.Hook[1].HookUnderOffset := L#115;
   Front.Hook[1].TelPos_1.TelPos := L#1;
   Front.Hook[2].HookOver := L#5560;
   Front.Hook[2].HookUnderOffset := L#115;
   Front.Hook[2].TelPos_1.TelPos := L#1;
   Front.Hook[3].HookOver := L#4415;
   Front.Hook[3].HookUnderOffset := L#115;
   Front.Hook[3].TelPos_1.TelPos := L#1;
   Front.Hook[4].HookOver := L#3260;
   Front.Hook[4].HookUnderOffset := L#115;
   Front.Hook[4].TelPos_1.TelPos := L#1;
   Front.Hook[5].HookOver := L#2115;
   Front.Hook[5].HookUnderOffset := L#115;
   Front.Hook[5].TelPos_1.TelPos := L#1;
   Rear.Hook[1].HookOver := L#6703;
   Rear.Hook[1].HookUnderOffset := L#115;
   Rear.Hook[1].TelPos_1.TelPos := L#2;
   Rear.Hook[2].HookOver := L#5560;
   Rear.Hook[2].HookUnderOffset := L#115;
   Rear.Hook[2].TelPos_1.TelPos := L#2;
   Rear.Hook[3].HookOver := L#4415;
   Rear.Hook[3].HookUnderOffset := L#115;
   Rear.Hook[3].TelPos_1.TelPos := L#2;
   Rear.Hook[4].HookOver := L#3260;
   Rear.Hook[4].HookUnderOffset := L#115;
   Rear.Hook[4].TelPos_1.TelPos := L#2;
   Rear.Hook[5].HookOver := L#2115;
   Rear.Hook[5].HookUnderOffset := L#115;
   Rear.Hook[5].TelPos_1.TelPos := L#2;
END_DATA_BLOCK

DATA_BLOCK "BR06_TR08"	// DB 263
VERSION : 0.1
  STRUCT
   Front : STRUCT
    Hook : ARRAY  [1 .. 10 ] OF UDT 102;
   END_STRUCT ;
   Rear : STRUCT
    Hook : ARRAY  [1 .. 10 ] OF UDT 102;
   END_STRUCT ;
  END_STRUCT ;	
BEGIN
   Front.Hook[1].HookOver := L#6703;
   Front.Hook[1].HookUnderOffset := L#115;
   Front.Hook[1].TelPos_1.TelPos := L#1;
   Front.Hook[2].HookOver := L#5560;
   Front.Hook[2].HookUnderOffset := L#115;
   Front.Hook[2].TelPos_1.TelPos := L#1;
   Front.Hook[3].HookOver := L#4415;
   Front.Hook[3].HookUnderOffset := L#115;
   Front.Hook[3].TelPos_1.TelPos := L#1;
   Front.Hook[4].HookOver := L#3260;
   Front.Hook[4].HookUnderOffset := L#115;
   Front.Hook[4].TelPos_1.TelPos := L#1;
   Front.Hook[5].HookOver := L#2115;
   Front.Hook[5].HookUnderOffset := L#115;
   Front.Hook[5].TelPos_1.TelPos := L#1;
   Rear.Hook[1].HookOver := L#6703;
   Rear.Hook[1].HookUnderOffset := L#115;
   Rear.Hook[1].TelPos_1.TelPos := L#2;
   Rear.Hook[2].HookOver := L#5560;
   Rear.Hook[2].HookUnderOffset := L#115;
   Rear.Hook[2].TelPos_1.TelPos := L#2;
   Rear.Hook[3].HookOver := L#4415;
   Rear.Hook[3].HookUnderOffset := L#115;
   Rear.Hook[3].TelPos_1.TelPos := L#2;
   Rear.Hook[4].HookOver := L#3260;
   Rear.Hook[4].HookUnderOffset := L#115;
   Rear.Hook[4].TelPos_1.TelPos := L#2;
   Rear.Hook[5].HookOver := L#2115;
   Rear.Hook[5].HookUnderOffset := L#115;
   Rear.Hook[5].TelPos_1.TelPos := L#2;
END_DATA_BLOCK

DATA_BLOCK "BR06_TR09"	// DB 264
VERSION : 0.1
  STRUCT
   Front : STRUCT
    Hook : ARRAY  [1 .. 10 ] OF UDT 102;
   END_STRUCT ;
   Rear : STRUCT
    Hook : ARRAY  [1 .. 10 ] OF UDT 102;
   END_STRUCT ;
  END_STRUCT ;	
BEGIN
END_DATA_BLOCK

DATA_BLOCK "BR06_TR10"	// DB 265
VERSION : 0.1
  STRUCT
   Front : STRUCT
    Hook : ARRAY  [1 .. 10 ] OF UDT 102;
   END_STRUCT ;
   Rear : STRUCT
    Hook : ARRAY  [1 .. 10 ] OF UDT 102;
   END_STRUCT ;
  END_STRUCT ;	
BEGIN
   Front.Hook[1].HookOver := L#6703;
   Front.Hook[1].HookUnderOffset := L#115;
   Front.Hook[2].HookOver := L#5560;
   Front.Hook[2].HookUnderOffset := L#115;
   Front.Hook[3].HookOver := L#4415;
   Front.Hook[3].HookUnderOffset := L#115;
   Front.Hook[3].TelPos_1.TelPos := L#1;
   Front.Hook[4].HookOver := L#3260;
   Front.Hook[4].HookUnderOffset := L#115;
   Front.Hook[4].TelPos_1.TelPos := L#1;
   Rear.Hook[1].HookOver := L#6703;
   Rear.Hook[1].HookUnderOffset := L#115;
   Rear.Hook[1].TelPos_1.TelPos := L#2;
   Rear.Hook[2].HookOver := L#5560;
   Rear.Hook[2].HookUnderOffset := L#115;
   Rear.Hook[2].TelPos_1.TelPos := L#2;
   Rear.Hook[3].HookOver := L#4415;
   Rear.Hook[3].HookUnderOffset := L#115;
   Rear.Hook[3].TelPos_1.TelPos := L#2;
   Rear.Hook[4].HookOver := L#3260;
   Rear.Hook[4].HookUnderOffset := L#115;
   Rear.Hook[4].TelPos_1.TelPos := L#2;
END_DATA_BLOCK

DATA_BLOCK "BR06_TR11"	// DB 266
VERSION : 0.1
  STRUCT
   Front : STRUCT
    Hook : ARRAY  [1 .. 10 ] OF UDT 102;
   END_STRUCT ;
   Rear : STRUCT
    Hook : ARRAY  [1 .. 10 ] OF UDT 102;
   END_STRUCT ;
  END_STRUCT ;	
BEGIN
END_DATA_BLOCK

DATA_BLOCK "BR07_TR01"	// DB 267
VERSION : 0.1
  STRUCT
   Front : STRUCT
    Hook : ARRAY  [1 .. 10 ] OF UDT 102;
   END_STRUCT ;
   Rear : STRUCT
    Hook : ARRAY  [1 .. 10 ] OF UDT 102;
   END_STRUCT ;
  END_STRUCT ;	
BEGIN
   Front.Hook[1].HookOver := L#6716;
   Front.Hook[1].HookUnderOffset := L#115;
   Front.Hook[1].TelPos_1.TelPos := L#1;
   Front.Hook[2].HookOver := L#5566;
   Front.Hook[2].HookUnderOffset := L#115;
   Front.Hook[2].TelPos_1.TelPos := L#1;
   Front.Hook[3].HookOver := L#4416;
   Front.Hook[3].HookUnderOffset := L#115;
   Front.Hook[3].TelPos_1.TelPos := L#1;
   Front.Hook[4].HookOver := L#3266;
   Front.Hook[4].HookUnderOffset := L#115;
   Front.Hook[4].TelPos_1.TelPos := L#1;
   Rear.Hook[1].HookOver := L#6716;
   Rear.Hook[1].HookUnderOffset := L#115;
   Rear.Hook[1].TelPos_1.TelPos := L#2;
   Rear.Hook[2].HookOver := L#5566;
   Rear.Hook[2].HookUnderOffset := L#115;
   Rear.Hook[2].TelPos_1.TelPos := L#2;
   Rear.Hook[3].HookOver := L#4416;
   Rear.Hook[3].HookUnderOffset := L#115;
   Rear.Hook[3].TelPos_1.TelPos := L#2;
   Rear.Hook[4].HookOver := L#3266;
   Rear.Hook[4].HookUnderOffset := L#115;
   Rear.Hook[4].TelPos_1.TelPos := L#2;
END_DATA_BLOCK

DATA_BLOCK "BR07_TR02"	// DB 268
VERSION : 0.1
  STRUCT
   Front : STRUCT
    Hook : ARRAY  [1 .. 10 ] OF UDT 102;
   END_STRUCT ;
   Rear : STRUCT
    Hook : ARRAY  [1 .. 10 ] OF UDT 102;
   END_STRUCT ;
  END_STRUCT ;	
BEGIN
   Front.Hook[1].HookOver := L#6703;
   Front.Hook[1].HookUnderOffset := L#115;
   Front.Hook[1].TelPos_1.TelPos := L#1;
   Front.Hook[2].HookOver := L#5560;
   Front.Hook[2].HookUnderOffset := L#115;
   Front.Hook[2].TelPos_1.TelPos := L#1;
   Front.Hook[3].HookOver := L#4415;
   Front.Hook[3].HookUnderOffset := L#115;
   Front.Hook[3].TelPos_1.TelPos := L#1;
   Front.Hook[4].HookOver := L#3260;
   Front.Hook[4].HookUnderOffset := L#115;
   Front.Hook[4].TelPos_1.TelPos := L#1;
   Front.Hook[5].HookOver := L#2115;
   Front.Hook[5].HookUnderOffset := L#115;
   Front.Hook[5].TelPos_1.TelPos := L#1;
   Rear.Hook[1].HookOver := L#6703;
   Rear.Hook[1].HookUnderOffset := L#115;
   Rear.Hook[1].TelPos_1.TelPos := L#2;
   Rear.Hook[2].HookOver := L#5560;
   Rear.Hook[2].HookUnderOffset := L#115;
   Rear.Hook[2].TelPos_1.TelPos := L#2;
   Rear.Hook[3].HookOver := L#4415;
   Rear.Hook[3].HookUnderOffset := L#115;
   Rear.Hook[3].TelPos_1.TelPos := L#2;
   Rear.Hook[4].HookOver := L#3260;
   Rear.Hook[4].HookUnderOffset := L#115;
   Rear.Hook[4].TelPos_1.TelPos := L#2;
   Rear.Hook[5].HookOver := L#2115;
   Rear.Hook[5].HookUnderOffset := L#115;
   Rear.Hook[5].TelPos_1.TelPos := L#2;
END_DATA_BLOCK

DATA_BLOCK "BR07_TR03"	// DB 269
VERSION : 0.1
  STRUCT
   Front : STRUCT
    Hook : ARRAY  [1 .. 10 ] OF UDT 102;
   END_STRUCT ;
   Rear : STRUCT
    Hook : ARRAY  [1 .. 10 ] OF UDT 102;
   END_STRUCT ;
  END_STRUCT ;	
BEGIN
   Front.Hook[1].HookOver := L#6703;
   Front.Hook[1].HookUnderOffset := L#115;
   Front.Hook[1].TelPos_1.TelPos := L#1;
   Front.Hook[2].HookOver := L#5560;
   Front.Hook[2].HookUnderOffset := L#115;
   Front.Hook[2].TelPos_1.TelPos := L#1;
   Front.Hook[3].HookOver := L#4415;
   Front.Hook[3].HookUnderOffset := L#115;
   Front.Hook[3].TelPos_1.TelPos := L#1;
   Front.Hook[4].HookOver := L#3260;
   Front.Hook[4].HookUnderOffset := L#115;
   Front.Hook[4].TelPos_1.TelPos := L#1;
   Front.Hook[5].HookOver := L#2115;
   Front.Hook[5].HookUnderOffset := L#115;
   Front.Hook[5].TelPos_1.TelPos := L#1;
   Rear.Hook[1].HookOver := L#6703;
   Rear.Hook[1].HookUnderOffset := L#115;
   Rear.Hook[1].TelPos_1.TelPos := L#2;
   Rear.Hook[2].HookOver := L#5560;
   Rear.Hook[2].HookUnderOffset := L#115;
   Rear.Hook[2].TelPos_1.TelPos := L#2;
   Rear.Hook[3].HookOver := L#4415;
   Rear.Hook[3].HookUnderOffset := L#115;
   Rear.Hook[3].TelPos_1.TelPos := L#2;
   Rear.Hook[4].HookOver := L#3260;
   Rear.Hook[4].HookUnderOffset := L#115;
   Rear.Hook[4].TelPos_1.TelPos := L#2;
   Rear.Hook[5].HookOver := L#2115;
   Rear.Hook[5].HookUnderOffset := L#115;
   Rear.Hook[5].TelPos_1.TelPos := L#2;
END_DATA_BLOCK

DATA_BLOCK "BR07_TR04"	// DB 270
VERSION : 0.1
  STRUCT
   Front : STRUCT
    Hook : ARRAY  [1 .. 10 ] OF UDT 102;
   END_STRUCT ;
   Rear : STRUCT
    Hook : ARRAY  [1 .. 10 ] OF UDT 102;
   END_STRUCT ;
  END_STRUCT ;	
BEGIN
   Front.Hook[1].HookOver := L#6703;
   Front.Hook[1].HookUnderOffset := L#115;
   Front.Hook[1].TelPos_1.TelPos := L#1;
   Front.Hook[2].HookOver := L#5560;
   Front.Hook[2].HookUnderOffset := L#115;
   Front.Hook[2].TelPos_1.TelPos := L#1;
   Front.Hook[3].HookOver := L#4415;
   Front.Hook[3].HookUnderOffset := L#115;
   Front.Hook[3].TelPos_1.TelPos := L#1;
   Front.Hook[4].HookOver := L#3260;
   Front.Hook[4].HookUnderOffset := L#115;
   Front.Hook[4].TelPos_1.TelPos := L#1;
   Front.Hook[5].HookOver := L#2115;
   Front.Hook[5].HookUnderOffset := L#115;
   Front.Hook[5].TelPos_1.TelPos := L#1;
   Rear.Hook[1].HookOver := L#6703;
   Rear.Hook[1].HookUnderOffset := L#115;
   Rear.Hook[1].TelPos_1.TelPos := L#2;
   Rear.Hook[2].HookOver := L#5560;
   Rear.Hook[2].HookUnderOffset := L#115;
   Rear.Hook[2].TelPos_1.TelPos := L#2;
   Rear.Hook[3].HookOver := L#4415;
   Rear.Hook[3].HookUnderOffset := L#115;
   Rear.Hook[3].TelPos_1.TelPos := L#2;
   Rear.Hook[4].HookOver := L#3260;
   Rear.Hook[4].HookUnderOffset := L#115;
   Rear.Hook[4].TelPos_1.TelPos := L#2;
   Rear.Hook[5].HookOver := L#2115;
   Rear.Hook[5].HookUnderOffset := L#115;
   Rear.Hook[5].TelPos_1.TelPos := L#2;
END_DATA_BLOCK

DATA_BLOCK "BR07_TR05"	// DB 271
VERSION : 0.1
  STRUCT
   Front : STRUCT
    Hook : ARRAY  [1 .. 10 ] OF UDT 102;
   END_STRUCT ;
   Rear : STRUCT
    Hook : ARRAY  [1 .. 10 ] OF UDT 102;
   END_STRUCT ;
  END_STRUCT ;	
BEGIN
   Front.Hook[1].HookOver := L#6703;
   Front.Hook[1].HookUnderOffset := L#115;
   Front.Hook[1].TelPos_1.TelPos := L#1;
   Front.Hook[2].HookOver := L#5560;
   Front.Hook[2].HookUnderOffset := L#115;
   Front.Hook[2].TelPos_1.TelPos := L#1;
   Front.Hook[3].HookOver := L#4415;
   Front.Hook[3].HookUnderOffset := L#115;
   Front.Hook[3].TelPos_1.TelPos := L#1;
   Front.Hook[4].HookOver := L#3260;
   Front.Hook[4].HookUnderOffset := L#115;
   Front.Hook[4].TelPos_1.TelPos := L#1;
   Front.Hook[5].HookOver := L#2115;
   Front.Hook[5].HookUnderOffset := L#115;
   Front.Hook[5].TelPos_1.TelPos := L#1;
   Rear.Hook[1].HookOver := L#6703;
   Rear.Hook[1].HookUnderOffset := L#115;
   Rear.Hook[1].TelPos_1.TelPos := L#2;
   Rear.Hook[2].HookOver := L#5560;
   Rear.Hook[2].HookUnderOffset := L#115;
   Rear.Hook[2].TelPos_1.TelPos := L#2;
   Rear.Hook[3].HookOver := L#4415;
   Rear.Hook[3].HookUnderOffset := L#115;
   Rear.Hook[3].TelPos_1.TelPos := L#2;
   Rear.Hook[4].HookOver := L#3260;
   Rear.Hook[4].HookUnderOffset := L#115;
   Rear.Hook[4].TelPos_1.TelPos := L#2;
   Rear.Hook[5].HookOver := L#2115;
   Rear.Hook[5].HookUnderOffset := L#115;
   Rear.Hook[5].TelPos_1.TelPos := L#2;
END_DATA_BLOCK

DATA_BLOCK "BR07_TR06"	// DB 272
VERSION : 0.1
  STRUCT
   Front : STRUCT
    Hook : ARRAY  [1 .. 10 ] OF UDT 102;
   END_STRUCT ;
   Rear : STRUCT
    Hook : ARRAY  [1 .. 10 ] OF UDT 102;
   END_STRUCT ;
  END_STRUCT ;	
BEGIN
   Front.Hook[1].HookOver := L#6703;
   Front.Hook[1].HookUnderOffset := L#115;
   Front.Hook[1].TelPos_1.TelPos := L#1;
   Front.Hook[2].HookOver := L#5560;
   Front.Hook[2].HookUnderOffset := L#115;
   Front.Hook[2].TelPos_1.TelPos := L#1;
   Front.Hook[3].HookOver := L#4415;
   Front.Hook[3].HookUnderOffset := L#115;
   Front.Hook[3].TelPos_1.TelPos := L#1;
   Front.Hook[4].HookOver := L#3260;
   Front.Hook[4].HookUnderOffset := L#115;
   Front.Hook[4].TelPos_1.TelPos := L#1;
   Front.Hook[5].HookOver := L#2115;
   Front.Hook[5].HookUnderOffset := L#115;
   Front.Hook[5].TelPos_1.TelPos := L#1;
   Rear.Hook[1].HookOver := L#6703;
   Rear.Hook[1].HookUnderOffset := L#115;
   Rear.Hook[1].TelPos_1.TelPos := L#2;
   Rear.Hook[2].HookOver := L#5560;
   Rear.Hook[2].HookUnderOffset := L#115;
   Rear.Hook[2].TelPos_1.TelPos := L#2;
   Rear.Hook[3].HookOver := L#4415;
   Rear.Hook[3].HookUnderOffset := L#115;
   Rear.Hook[3].TelPos_1.TelPos := L#2;
   Rear.Hook[4].HookOver := L#3260;
   Rear.Hook[4].HookUnderOffset := L#115;
   Rear.Hook[4].TelPos_1.TelPos := L#2;
   Rear.Hook[5].HookOver := L#2115;
   Rear.Hook[5].HookUnderOffset := L#115;
   Rear.Hook[5].TelPos_1.TelPos := L#2;
END_DATA_BLOCK

DATA_BLOCK "BR07_TR07"	// DB 273
VERSION : 0.1
  STRUCT
   Front : STRUCT
    Hook : ARRAY  [1 .. 10 ] OF UDT 102;
   END_STRUCT ;
   Rear : STRUCT
    Hook : ARRAY  [1 .. 10 ] OF UDT 102;
   END_STRUCT ;
  END_STRUCT ;	
BEGIN
   Front.Hook[1].HookOver := L#6703;
   Front.Hook[1].HookUnderOffset := L#115;
   Front.Hook[1].TelPos_1.TelPos := L#1;
   Front.Hook[2].HookOver := L#5560;
   Front.Hook[2].HookUnderOffset := L#115;
   Front.Hook[2].TelPos_1.TelPos := L#1;
   Front.Hook[3].HookOver := L#4415;
   Front.Hook[3].HookUnderOffset := L#115;
   Front.Hook[3].TelPos_1.TelPos := L#1;
   Front.Hook[4].HookOver := L#3260;
   Front.Hook[4].HookUnderOffset := L#115;
   Front.Hook[4].TelPos_1.TelPos := L#1;
   Front.Hook[5].HookOver := L#2115;
   Front.Hook[5].HookUnderOffset := L#115;
   Front.Hook[5].TelPos_1.TelPos := L#1;
   Rear.Hook[1].HookOver := L#6703;
   Rear.Hook[1].HookUnderOffset := L#115;
   Rear.Hook[1].TelPos_1.TelPos := L#2;
   Rear.Hook[2].HookOver := L#5560;
   Rear.Hook[2].HookUnderOffset := L#115;
   Rear.Hook[2].TelPos_1.TelPos := L#2;
   Rear.Hook[3].HookOver := L#4415;
   Rear.Hook[3].HookUnderOffset := L#115;
   Rear.Hook[3].TelPos_1.TelPos := L#2;
   Rear.Hook[4].HookOver := L#3260;
   Rear.Hook[4].HookUnderOffset := L#115;
   Rear.Hook[4].TelPos_1.TelPos := L#2;
   Rear.Hook[5].HookOver := L#2115;
   Rear.Hook[5].HookUnderOffset := L#115;
   Rear.Hook[5].TelPos_1.TelPos := L#2;
END_DATA_BLOCK

DATA_BLOCK "BR07_TR08"	// DB 274
VERSION : 0.1
  STRUCT
   Front : STRUCT
    Hook : ARRAY  [1 .. 10 ] OF UDT 102;
   END_STRUCT ;
   Rear : STRUCT
    Hook : ARRAY  [1 .. 10 ] OF UDT 102;
   END_STRUCT ;
  END_STRUCT ;	
BEGIN
   Front.Hook[1].HookOver := L#6703;
   Front.Hook[1].HookUnderOffset := L#115;
   Front.Hook[1].TelPos_1.TelPos := L#1;
   Front.Hook[2].HookOver := L#5560;
   Front.Hook[2].HookUnderOffset := L#115;
   Front.Hook[2].TelPos_1.TelPos := L#1;
   Front.Hook[3].HookOver := L#4415;
   Front.Hook[3].HookUnderOffset := L#115;
   Front.Hook[3].TelPos_1.TelPos := L#1;
   Front.Hook[4].HookOver := L#3260;
   Front.Hook[4].HookUnderOffset := L#115;
   Front.Hook[4].TelPos_1.TelPos := L#1;
   Front.Hook[5].HookOver := L#2115;
   Front.Hook[5].HookUnderOffset := L#115;
   Front.Hook[5].TelPos_1.TelPos := L#1;
   Rear.Hook[1].HookOver := L#6703;
   Rear.Hook[1].HookUnderOffset := L#115;
   Rear.Hook[1].TelPos_1.TelPos := L#2;
   Rear.Hook[2].HookOver := L#5560;
   Rear.Hook[2].HookUnderOffset := L#115;
   Rear.Hook[2].TelPos_1.TelPos := L#2;
   Rear.Hook[3].HookOver := L#4415;
   Rear.Hook[3].HookUnderOffset := L#115;
   Rear.Hook[3].TelPos_1.TelPos := L#2;
   Rear.Hook[4].HookOver := L#3260;
   Rear.Hook[4].HookUnderOffset := L#115;
   Rear.Hook[4].TelPos_1.TelPos := L#2;
   Rear.Hook[5].HookOver := L#2115;
   Rear.Hook[5].HookUnderOffset := L#115;
   Rear.Hook[5].TelPos_1.TelPos := L#2;
END_DATA_BLOCK

DATA_BLOCK "BR07_TR09"	// DB 275
VERSION : 0.1
  STRUCT
   Front : STRUCT
    Hook : ARRAY  [1 .. 10 ] OF UDT 102;
   END_STRUCT ;
   Rear : STRUCT
    Hook : ARRAY  [1 .. 10 ] OF UDT 102;
   END_STRUCT ;
  END_STRUCT ;	
BEGIN
END_DATA_BLOCK

DATA_BLOCK "BR07_TR10"	// DB 276
VERSION : 0.1
  STRUCT
   Front : STRUCT
    Hook : ARRAY  [1 .. 10 ] OF UDT 102;
   END_STRUCT ;
   Rear : STRUCT
    Hook : ARRAY  [1 .. 10 ] OF UDT 102;
   END_STRUCT ;
  END_STRUCT ;	
BEGIN
   Front.Hook[1].HookOver := L#6703;
   Front.Hook[1].HookUnderOffset := L#115;
   Front.Hook[2].HookOver := L#5560;
   Front.Hook[2].HookUnderOffset := L#115;
   Front.Hook[3].HookOver := L#4415;
   Front.Hook[3].HookUnderOffset := L#115;
   Front.Hook[3].TelPos_1.TelPos := L#1;
   Front.Hook[4].HookOver := L#3260;
   Front.Hook[4].HookUnderOffset := L#115;
   Front.Hook[4].TelPos_1.TelPos := L#1;
   Rear.Hook[1].HookOver := L#6703;
   Rear.Hook[1].HookUnderOffset := L#115;
   Rear.Hook[1].TelPos_1.TelPos := L#2;
   Rear.Hook[2].HookOver := L#5560;
   Rear.Hook[2].HookUnderOffset := L#115;
   Rear.Hook[2].TelPos_1.TelPos := L#2;
   Rear.Hook[3].HookOver := L#4415;
   Rear.Hook[3].HookUnderOffset := L#115;
   Rear.Hook[3].TelPos_1.TelPos := L#2;
   Rear.Hook[4].HookOver := L#3260;
   Rear.Hook[4].HookUnderOffset := L#115;
   Rear.Hook[4].TelPos_1.TelPos := L#2;
END_DATA_BLOCK

DATA_BLOCK "BR07_TR11"	// DB 277
VERSION : 0.1
  STRUCT
   Front : STRUCT
    Hook : ARRAY  [1 .. 10 ] OF UDT 102;
   END_STRUCT ;
   Rear : STRUCT
    Hook : ARRAY  [1 .. 10 ] OF UDT 102;
   END_STRUCT ;
  END_STRUCT ;	
BEGIN
END_DATA_BLOCK

DATA_BLOCK "BR08_TR01"	// DB 278
VERSION : 0.1
  STRUCT
   Front : STRUCT
    Hook : ARRAY  [1 .. 10 ] OF UDT 102;
   END_STRUCT ;
   Rear : STRUCT
    Hook : ARRAY  [1 .. 10 ] OF UDT 102;
   END_STRUCT ;
  END_STRUCT ;	
BEGIN
   Front.Hook[1].HookOver := L#6650;
   Front.Hook[1].HookUnderOffset := L#115;
   Front.Hook[1].TelPos_1.TelPos := L#1;
   Front.Hook[2].HookOver := L#5566;
   Front.Hook[2].HookUnderOffset := L#115;
   Front.Hook[2].TelPos_1.TelPos := L#1;
   Front.Hook[3].HookOver := L#4416;
   Front.Hook[3].HookUnderOffset := L#115;
   Front.Hook[3].TelPos_1.TelPos := L#1;
   Front.Hook[4].HookOver := L#3266;
   Front.Hook[4].HookUnderOffset := L#115;
   Front.Hook[4].TelPos_1.TelPos := L#1;
   Rear.Hook[1].HookOver := L#6716;
   Rear.Hook[1].HookUnderOffset := L#115;
   Rear.Hook[1].TelPos_1.TelPos := L#2;
   Rear.Hook[2].HookOver := L#5566;
   Rear.Hook[2].HookUnderOffset := L#115;
   Rear.Hook[2].TelPos_1.TelPos := L#2;
   Rear.Hook[3].HookOver := L#4416;
   Rear.Hook[3].HookUnderOffset := L#115;
   Rear.Hook[3].TelPos_1.TelPos := L#2;
   Rear.Hook[4].HookOver := L#3266;
   Rear.Hook[4].HookUnderOffset := L#115;
   Rear.Hook[4].TelPos_1.TelPos := L#2;
END_DATA_BLOCK

DATA_BLOCK "BR08_TR02"	// DB 279
VERSION : 0.1
  STRUCT
   Front : STRUCT
    Hook : ARRAY  [1 .. 10 ] OF UDT 102;
   END_STRUCT ;
   Rear : STRUCT
    Hook : ARRAY  [1 .. 10 ] OF UDT 102;
   END_STRUCT ;
  END_STRUCT ;	
BEGIN
   Front.Hook[1].HookOver := L#6703;
   Front.Hook[1].HookUnderOffset := L#115;
   Front.Hook[1].TelPos_1.TelPos := L#1;
   Front.Hook[2].HookOver := L#5560;
   Front.Hook[2].HookUnderOffset := L#115;
   Front.Hook[2].TelPos_1.TelPos := L#1;
   Front.Hook[3].HookOver := L#4415;
   Front.Hook[3].HookUnderOffset := L#115;
   Front.Hook[3].TelPos_1.TelPos := L#1;
   Front.Hook[4].HookOver := L#3260;
   Front.Hook[4].HookUnderOffset := L#115;
   Front.Hook[4].TelPos_1.TelPos := L#1;
   Front.Hook[5].HookOver := L#2115;
   Front.Hook[5].HookUnderOffset := L#115;
   Front.Hook[5].TelPos_1.TelPos := L#1;
   Rear.Hook[1].HookOver := L#6703;
   Rear.Hook[1].HookUnderOffset := L#115;
   Rear.Hook[1].TelPos_1.TelPos := L#2;
   Rear.Hook[2].HookOver := L#5560;
   Rear.Hook[2].HookUnderOffset := L#115;
   Rear.Hook[2].TelPos_1.TelPos := L#2;
   Rear.Hook[3].HookOver := L#4415;
   Rear.Hook[3].HookUnderOffset := L#115;
   Rear.Hook[3].TelPos_1.TelPos := L#2;
   Rear.Hook[4].HookOver := L#3260;
   Rear.Hook[4].HookUnderOffset := L#115;
   Rear.Hook[4].TelPos_1.TelPos := L#2;
   Rear.Hook[5].HookOver := L#2115;
   Rear.Hook[5].HookUnderOffset := L#115;
   Rear.Hook[5].TelPos_1.TelPos := L#2;
END_DATA_BLOCK

DATA_BLOCK "BR08_TR03"	// DB 280
VERSION : 0.1
  STRUCT
   Front : STRUCT
    Hook : ARRAY  [1 .. 10 ] OF UDT 102;
   END_STRUCT ;
   Rear : STRUCT
    Hook : ARRAY  [1 .. 10 ] OF UDT 102;
   END_STRUCT ;
  END_STRUCT ;	
BEGIN
   Front.Hook[1].HookOver := L#6703;
   Front.Hook[1].HookUnderOffset := L#115;
   Front.Hook[1].TelPos_1.TelPos := L#1;
   Front.Hook[2].HookOver := L#5560;
   Front.Hook[2].HookUnderOffset := L#115;
   Front.Hook[2].TelPos_1.TelPos := L#1;
   Front.Hook[3].HookOver := L#4415;
   Front.Hook[3].HookUnderOffset := L#115;
   Front.Hook[3].TelPos_1.TelPos := L#1;
   Front.Hook[4].HookOver := L#3260;
   Front.Hook[4].HookUnderOffset := L#115;
   Front.Hook[4].TelPos_1.TelPos := L#1;
   Front.Hook[5].HookOver := L#2115;
   Front.Hook[5].HookUnderOffset := L#115;
   Front.Hook[5].TelPos_1.TelPos := L#1;
   Rear.Hook[1].HookOver := L#6703;
   Rear.Hook[1].HookUnderOffset := L#115;
   Rear.Hook[1].TelPos_1.TelPos := L#2;
   Rear.Hook[2].HookOver := L#5560;
   Rear.Hook[2].HookUnderOffset := L#115;
   Rear.Hook[2].TelPos_1.TelPos := L#2;
   Rear.Hook[3].HookOver := L#4415;
   Rear.Hook[3].HookUnderOffset := L#115;
   Rear.Hook[3].TelPos_1.TelPos := L#2;
   Rear.Hook[4].HookOver := L#3260;
   Rear.Hook[4].HookUnderOffset := L#115;
   Rear.Hook[4].TelPos_1.TelPos := L#2;
   Rear.Hook[5].HookOver := L#2115;
   Rear.Hook[5].HookUnderOffset := L#115;
   Rear.Hook[5].TelPos_1.TelPos := L#2;
END_DATA_BLOCK

DATA_BLOCK "BR08_TR04"	// DB 281
VERSION : 0.1
  STRUCT
   Front : STRUCT
    Hook : ARRAY  [1 .. 10 ] OF UDT 102;
   END_STRUCT ;
   Rear : STRUCT
    Hook : ARRAY  [1 .. 10 ] OF UDT 102;
   END_STRUCT ;
  END_STRUCT ;	
BEGIN
   Front.Hook[1].HookOver := L#6703;
   Front.Hook[1].HookUnderOffset := L#115;
   Front.Hook[1].TelPos_1.TelPos := L#1;
   Front.Hook[2].HookOver := L#5560;
   Front.Hook[2].HookUnderOffset := L#115;
   Front.Hook[2].TelPos_1.TelPos := L#1;
   Front.Hook[3].HookOver := L#4415;
   Front.Hook[3].HookUnderOffset := L#115;
   Front.Hook[3].TelPos_1.TelPos := L#1;
   Front.Hook[4].HookOver := L#3260;
   Front.Hook[4].HookUnderOffset := L#115;
   Front.Hook[4].TelPos_1.TelPos := L#1;
   Front.Hook[5].HookOver := L#2115;
   Front.Hook[5].HookUnderOffset := L#115;
   Front.Hook[5].TelPos_1.TelPos := L#1;
   Rear.Hook[1].HookOver := L#6703;
   Rear.Hook[1].HookUnderOffset := L#115;
   Rear.Hook[1].TelPos_1.TelPos := L#2;
   Rear.Hook[2].HookOver := L#5560;
   Rear.Hook[2].HookUnderOffset := L#115;
   Rear.Hook[2].TelPos_1.TelPos := L#2;
   Rear.Hook[3].HookOver := L#4415;
   Rear.Hook[3].HookUnderOffset := L#115;
   Rear.Hook[3].TelPos_1.TelPos := L#2;
   Rear.Hook[4].HookOver := L#3260;
   Rear.Hook[4].HookUnderOffset := L#115;
   Rear.Hook[4].TelPos_1.TelPos := L#2;
   Rear.Hook[5].HookOver := L#2115;
   Rear.Hook[5].HookUnderOffset := L#115;
   Rear.Hook[5].TelPos_1.TelPos := L#2;
END_DATA_BLOCK

DATA_BLOCK "BR08_TR05"	// DB 282
VERSION : 0.1
  STRUCT
   Front : STRUCT
    Hook : ARRAY  [1 .. 10 ] OF UDT 102;
   END_STRUCT ;
   Rear : STRUCT
    Hook : ARRAY  [1 .. 10 ] OF UDT 102;
   END_STRUCT ;
  END_STRUCT ;	
BEGIN
   Front.Hook[1].HookOver := L#6703;
   Front.Hook[1].HookUnderOffset := L#115;
   Front.Hook[1].TelPos_1.TelPos := L#1;
   Front.Hook[2].HookOver := L#5560;
   Front.Hook[2].HookUnderOffset := L#115;
   Front.Hook[2].TelPos_1.TelPos := L#1;
   Front.Hook[3].HookOver := L#4415;
   Front.Hook[3].HookUnderOffset := L#115;
   Front.Hook[3].TelPos_1.TelPos := L#1;
   Front.Hook[4].HookOver := L#3260;
   Front.Hook[4].HookUnderOffset := L#115;
   Front.Hook[4].TelPos_1.TelPos := L#1;
   Front.Hook[5].HookOver := L#2115;
   Front.Hook[5].HookUnderOffset := L#115;
   Front.Hook[5].TelPos_1.TelPos := L#1;
   Rear.Hook[1].HookOver := L#6703;
   Rear.Hook[1].HookUnderOffset := L#115;
   Rear.Hook[1].TelPos_1.TelPos := L#2;
   Rear.Hook[2].HookOver := L#5560;
   Rear.Hook[2].HookUnderOffset := L#115;
   Rear.Hook[2].TelPos_1.TelPos := L#2;
   Rear.Hook[3].HookOver := L#4415;
   Rear.Hook[3].HookUnderOffset := L#115;
   Rear.Hook[3].TelPos_1.TelPos := L#2;
   Rear.Hook[4].HookOver := L#3260;
   Rear.Hook[4].HookUnderOffset := L#115;
   Rear.Hook[4].TelPos_1.TelPos := L#2;
   Rear.Hook[5].HookOver := L#2115;
   Rear.Hook[5].HookUnderOffset := L#115;
   Rear.Hook[5].TelPos_1.TelPos := L#2;
END_DATA_BLOCK

DATA_BLOCK "BR08_TR06"	// DB 283
VERSION : 0.1
  STRUCT
   Front : STRUCT
    Hook : ARRAY  [1 .. 10 ] OF UDT 102;
   END_STRUCT ;
   Rear : STRUCT
    Hook : ARRAY  [1 .. 10 ] OF UDT 102;
   END_STRUCT ;
  END_STRUCT ;	
BEGIN
   Front.Hook[1].HookOver := L#6703;
   Front.Hook[1].HookUnderOffset := L#115;
   Front.Hook[1].TelPos_1.TelPos := L#1;
   Front.Hook[2].HookOver := L#5560;
   Front.Hook[2].HookUnderOffset := L#115;
   Front.Hook[2].TelPos_1.TelPos := L#1;
   Front.Hook[3].HookOver := L#4415;
   Front.Hook[3].HookUnderOffset := L#115;
   Front.Hook[3].TelPos_1.TelPos := L#1;
   Front.Hook[4].HookOver := L#3260;
   Front.Hook[4].HookUnderOffset := L#115;
   Front.Hook[4].TelPos_1.TelPos := L#1;
   Front.Hook[5].HookOver := L#2115;
   Front.Hook[5].HookUnderOffset := L#115;
   Front.Hook[5].TelPos_1.TelPos := L#1;
   Rear.Hook[1].HookOver := L#6703;
   Rear.Hook[1].HookUnderOffset := L#115;
   Rear.Hook[1].TelPos_1.TelPos := L#2;
   Rear.Hook[2].HookOver := L#5560;
   Rear.Hook[2].HookUnderOffset := L#115;
   Rear.Hook[2].TelPos_1.TelPos := L#2;
   Rear.Hook[3].HookOver := L#4415;
   Rear.Hook[3].HookUnderOffset := L#115;
   Rear.Hook[3].TelPos_1.TelPos := L#2;
   Rear.Hook[4].HookOver := L#3260;
   Rear.Hook[4].HookUnderOffset := L#115;
   Rear.Hook[4].TelPos_1.TelPos := L#2;
   Rear.Hook[5].HookOver := L#2115;
   Rear.Hook[5].HookUnderOffset := L#115;
   Rear.Hook[5].TelPos_1.TelPos := L#2;
END_DATA_BLOCK

DATA_BLOCK "BR08_TR07"	// DB 284
VERSION : 0.1
  STRUCT
   Front : STRUCT
    Hook : ARRAY  [1 .. 10 ] OF UDT 102;
   END_STRUCT ;
   Rear : STRUCT
    Hook : ARRAY  [1 .. 10 ] OF UDT 102;
   END_STRUCT ;
  END_STRUCT ;	
BEGIN
   Front.Hook[1].HookOver := L#6703;
   Front.Hook[1].HookUnderOffset := L#115;
   Front.Hook[1].TelPos_1.TelPos := L#1;
   Front.Hook[2].HookOver := L#5560;
   Front.Hook[2].HookUnderOffset := L#115;
   Front.Hook[2].TelPos_1.TelPos := L#1;
   Front.Hook[3].HookOver := L#4415;
   Front.Hook[3].HookUnderOffset := L#115;
   Front.Hook[3].TelPos_1.TelPos := L#1;
   Front.Hook[4].HookOver := L#3260;
   Front.Hook[4].HookUnderOffset := L#115;
   Front.Hook[4].TelPos_1.TelPos := L#1;
   Front.Hook[5].HookOver := L#2115;
   Front.Hook[5].HookUnderOffset := L#115;
   Front.Hook[5].TelPos_1.TelPos := L#1;
   Rear.Hook[1].HookOver := L#6703;
   Rear.Hook[1].HookUnderOffset := L#115;
   Rear.Hook[1].TelPos_1.TelPos := L#2;
   Rear.Hook[2].HookOver := L#5560;
   Rear.Hook[2].HookUnderOffset := L#115;
   Rear.Hook[2].TelPos_1.TelPos := L#2;
   Rear.Hook[3].HookOver := L#4415;
   Rear.Hook[3].HookUnderOffset := L#115;
   Rear.Hook[3].TelPos_1.TelPos := L#2;
   Rear.Hook[4].HookOver := L#3260;
   Rear.Hook[4].HookUnderOffset := L#115;
   Rear.Hook[4].TelPos_1.TelPos := L#2;
   Rear.Hook[5].HookOver := L#2115;
   Rear.Hook[5].HookUnderOffset := L#115;
   Rear.Hook[5].TelPos_1.TelPos := L#2;
END_DATA_BLOCK

DATA_BLOCK "BR08_TR08"	// DB 285
VERSION : 0.1
  STRUCT
   Front : STRUCT
    Hook : ARRAY  [1 .. 10 ] OF UDT 102;
   END_STRUCT ;
   Rear : STRUCT
    Hook : ARRAY  [1 .. 10 ] OF UDT 102;
   END_STRUCT ;
  END_STRUCT ;	
BEGIN
   Front.Hook[1].HookOver := L#6703;
   Front.Hook[1].HookUnderOffset := L#115;
   Front.Hook[1].TelPos_1.TelPos := L#1;
   Front.Hook[2].HookOver := L#5560;
   Front.Hook[2].HookUnderOffset := L#115;
   Front.Hook[2].TelPos_1.TelPos := L#1;
   Front.Hook[3].HookOver := L#4415;
   Front.Hook[3].HookUnderOffset := L#115;
   Front.Hook[3].TelPos_1.TelPos := L#1;
   Front.Hook[4].HookOver := L#3260;
   Front.Hook[4].HookUnderOffset := L#115;
   Front.Hook[4].TelPos_1.TelPos := L#1;
   Front.Hook[5].HookOver := L#2115;
   Front.Hook[5].HookUnderOffset := L#115;
   Front.Hook[5].TelPos_1.TelPos := L#1;
   Rear.Hook[1].HookOver := L#6703;
   Rear.Hook[1].HookUnderOffset := L#115;
   Rear.Hook[1].TelPos_1.TelPos := L#2;
   Rear.Hook[2].HookOver := L#5560;
   Rear.Hook[2].HookUnderOffset := L#115;
   Rear.Hook[2].TelPos_1.TelPos := L#2;
   Rear.Hook[3].HookOver := L#4415;
   Rear.Hook[3].HookUnderOffset := L#115;
   Rear.Hook[3].TelPos_1.TelPos := L#2;
   Rear.Hook[4].HookOver := L#3260;
   Rear.Hook[4].HookUnderOffset := L#115;
   Rear.Hook[4].TelPos_1.TelPos := L#2;
   Rear.Hook[5].HookOver := L#2115;
   Rear.Hook[5].HookUnderOffset := L#115;
   Rear.Hook[5].TelPos_1.TelPos := L#2;
END_DATA_BLOCK

DATA_BLOCK "BR08_TR09"	// DB 286
VERSION : 0.1
  STRUCT
   Front : STRUCT
    Hook : ARRAY  [1 .. 10 ] OF UDT 102;
   END_STRUCT ;
   Rear : STRUCT
    Hook : ARRAY  [1 .. 10 ] OF UDT 102;
   END_STRUCT ;
  END_STRUCT ;	
BEGIN
END_DATA_BLOCK

DATA_BLOCK "BR08_TR10"	// DB 287
VERSION : 0.1
  STRUCT
   Front : STRUCT
    Hook : ARRAY  [1 .. 10 ] OF UDT 102;
   END_STRUCT ;
   Rear : STRUCT
    Hook : ARRAY  [1 .. 10 ] OF UDT 102;
   END_STRUCT ;
  END_STRUCT ;	
BEGIN
   Front.Hook[1].HookOver := L#6703;
   Front.Hook[1].HookUnderOffset := L#115;
   Front.Hook[2].HookOver := L#5560;
   Front.Hook[2].HookUnderOffset := L#115;
   Front.Hook[3].HookOver := L#4415;
   Front.Hook[3].HookUnderOffset := L#115;
   Front.Hook[3].TelPos_1.TelPos := L#1;
   Front.Hook[4].HookOver := L#3260;
   Front.Hook[4].HookUnderOffset := L#115;
   Front.Hook[4].TelPos_1.TelPos := L#1;
   Rear.Hook[1].HookOver := L#6703;
   Rear.Hook[1].HookUnderOffset := L#115;
   Rear.Hook[1].TelPos_1.TelPos := L#2;
   Rear.Hook[2].HookOver := L#5560;
   Rear.Hook[2].HookUnderOffset := L#115;
   Rear.Hook[2].TelPos_1.TelPos := L#2;
   Rear.Hook[3].HookOver := L#4415;
   Rear.Hook[3].HookUnderOffset := L#115;
   Rear.Hook[3].TelPos_1.TelPos := L#2;
   Rear.Hook[4].HookOver := L#3260;
   Rear.Hook[4].HookUnderOffset := L#115;
   Rear.Hook[4].TelPos_1.TelPos := L#2;
END_DATA_BLOCK

DATA_BLOCK "BR08_TR11"	// DB 288
VERSION : 0.1
  STRUCT
   Front : STRUCT
    Hook : ARRAY  [1 .. 10 ] OF UDT 102;
   END_STRUCT ;
   Rear : STRUCT
    Hook : ARRAY  [1 .. 10 ] OF UDT 102;
   END_STRUCT ;
  END_STRUCT ;	
BEGIN
END_DATA_BLOCK

DATA_BLOCK "BR09_TR01"	// DB 289
VERSION : 0.1
  STRUCT
   Front : STRUCT
    Hook : ARRAY  [1 .. 10 ] OF UDT 102;
   END_STRUCT ;
   Rear : STRUCT
    Hook : ARRAY  [1 .. 10 ] OF UDT 102;
   END_STRUCT ;
  END_STRUCT ;	
BEGIN
   Front.Hook[1].HookOver := L#6716;
   Front.Hook[1].HookUnderOffset := L#115;
   Front.Hook[1].TelPos_1.TelPos := L#1;
   Front.Hook[2].HookOver := L#5566;
   Front.Hook[2].HookUnderOffset := L#115;
   Front.Hook[2].TelPos_1.TelPos := L#1;
   Front.Hook[3].HookOver := L#4416;
   Front.Hook[3].HookUnderOffset := L#115;
   Front.Hook[3].TelPos_1.TelPos := L#1;
   Front.Hook[4].HookOver := L#3266;
   Front.Hook[4].HookUnderOffset := L#115;
   Front.Hook[4].TelPos_1.TelPos := L#1;
   Rear.Hook[1].HookOver := L#6716;
   Rear.Hook[1].HookUnderOffset := L#115;
   Rear.Hook[1].TelPos_1.TelPos := L#2;
   Rear.Hook[2].HookOver := L#5566;
   Rear.Hook[2].HookUnderOffset := L#115;
   Rear.Hook[2].TelPos_1.TelPos := L#2;
   Rear.Hook[3].HookOver := L#4416;
   Rear.Hook[3].HookUnderOffset := L#115;
   Rear.Hook[3].TelPos_1.TelPos := L#2;
   Rear.Hook[4].HookOver := L#3266;
   Rear.Hook[4].HookUnderOffset := L#115;
   Rear.Hook[4].TelPos_1.TelPos := L#2;
END_DATA_BLOCK

DATA_BLOCK "BR09_TR02"	// DB 290
VERSION : 0.1
  STRUCT
   Front : STRUCT
    Hook : ARRAY  [1 .. 10 ] OF UDT 102;
   END_STRUCT ;
   Rear : STRUCT
    Hook : ARRAY  [1 .. 10 ] OF UDT 102;
   END_STRUCT ;
  END_STRUCT ;	
BEGIN
   Front.Hook[1].HookOver := L#6703;
   Front.Hook[1].HookUnderOffset := L#115;
   Front.Hook[1].TelPos_1.TelPos := L#1;
   Front.Hook[2].HookOver := L#5560;
   Front.Hook[2].HookUnderOffset := L#115;
   Front.Hook[2].TelPos_1.TelPos := L#1;
   Front.Hook[3].HookOver := L#4415;
   Front.Hook[3].HookUnderOffset := L#115;
   Front.Hook[3].TelPos_1.TelPos := L#1;
   Front.Hook[4].HookOver := L#3260;
   Front.Hook[4].HookUnderOffset := L#115;
   Front.Hook[4].TelPos_1.TelPos := L#1;
   Front.Hook[5].HookOver := L#2115;
   Front.Hook[5].HookUnderOffset := L#115;
   Front.Hook[5].TelPos_1.TelPos := L#1;
   Rear.Hook[1].HookOver := L#6703;
   Rear.Hook[1].HookUnderOffset := L#115;
   Rear.Hook[1].TelPos_1.TelPos := L#2;
   Rear.Hook[2].HookOver := L#5560;
   Rear.Hook[2].HookUnderOffset := L#115;
   Rear.Hook[2].TelPos_1.TelPos := L#2;
   Rear.Hook[3].HookOver := L#4415;
   Rear.Hook[3].HookUnderOffset := L#115;
   Rear.Hook[3].TelPos_1.TelPos := L#2;
   Rear.Hook[4].HookOver := L#3260;
   Rear.Hook[4].HookUnderOffset := L#115;
   Rear.Hook[4].TelPos_1.TelPos := L#2;
   Rear.Hook[5].HookOver := L#2115;
   Rear.Hook[5].HookUnderOffset := L#115;
   Rear.Hook[5].TelPos_1.TelPos := L#2;
END_DATA_BLOCK

DATA_BLOCK "BR09_TR03"	// DB 291
VERSION : 0.1
  STRUCT
   Front : STRUCT
    Hook : ARRAY  [1 .. 10 ] OF UDT 102;
   END_STRUCT ;
   Rear : STRUCT
    Hook : ARRAY  [1 .. 10 ] OF UDT 102;
   END_STRUCT ;
  END_STRUCT ;	
BEGIN
   Front.Hook[1].HookOver := L#6703;
   Front.Hook[1].HookUnderOffset := L#115;
   Front.Hook[1].TelPos_1.TelPos := L#1;
   Front.Hook[2].HookOver := L#5560;
   Front.Hook[2].HookUnderOffset := L#115;
   Front.Hook[2].TelPos_1.TelPos := L#1;
   Front.Hook[3].HookOver := L#4415;
   Front.Hook[3].HookUnderOffset := L#115;
   Front.Hook[3].TelPos_1.TelPos := L#1;
   Front.Hook[4].HookOver := L#3260;
   Front.Hook[4].HookUnderOffset := L#115;
   Front.Hook[4].TelPos_1.TelPos := L#1;
   Front.Hook[5].HookOver := L#2115;
   Front.Hook[5].HookUnderOffset := L#115;
   Front.Hook[5].TelPos_1.TelPos := L#1;
   Rear.Hook[1].HookOver := L#6703;
   Rear.Hook[1].HookUnderOffset := L#115;
   Rear.Hook[1].TelPos_1.TelPos := L#2;
   Rear.Hook[2].HookOver := L#5560;
   Rear.Hook[2].HookUnderOffset := L#115;
   Rear.Hook[2].TelPos_1.TelPos := L#2;
   Rear.Hook[3].HookOver := L#4415;
   Rear.Hook[3].HookUnderOffset := L#115;
   Rear.Hook[3].TelPos_1.TelPos := L#2;
   Rear.Hook[4].HookOver := L#3260;
   Rear.Hook[4].HookUnderOffset := L#115;
   Rear.Hook[4].TelPos_1.TelPos := L#2;
   Rear.Hook[5].HookOver := L#2115;
   Rear.Hook[5].HookUnderOffset := L#115;
   Rear.Hook[5].TelPos_1.TelPos := L#2;
END_DATA_BLOCK

DATA_BLOCK "BR09_TR04"	// DB 292
VERSION : 0.1
  STRUCT
   Front : STRUCT
    Hook : ARRAY  [1 .. 10 ] OF UDT 102;
   END_STRUCT ;
   Rear : STRUCT
    Hook : ARRAY  [1 .. 10 ] OF UDT 102;
   END_STRUCT ;
  END_STRUCT ;	
BEGIN
   Front.Hook[1].HookOver := L#6703;
   Front.Hook[1].HookUnderOffset := L#115;
   Front.Hook[1].TelPos_1.TelPos := L#1;
   Front.Hook[2].HookOver := L#5560;
   Front.Hook[2].HookUnderOffset := L#115;
   Front.Hook[2].TelPos_1.TelPos := L#1;
   Front.Hook[3].HookOver := L#4415;
   Front.Hook[3].HookUnderOffset := L#115;
   Front.Hook[3].TelPos_1.TelPos := L#1;
   Front.Hook[4].HookOver := L#3260;
   Front.Hook[4].HookUnderOffset := L#115;
   Front.Hook[4].TelPos_1.TelPos := L#1;
   Front.Hook[5].HookOver := L#2115;
   Front.Hook[5].HookUnderOffset := L#115;
   Front.Hook[5].TelPos_1.TelPos := L#1;
   Rear.Hook[1].HookOver := L#6703;
   Rear.Hook[1].HookUnderOffset := L#115;
   Rear.Hook[1].TelPos_1.TelPos := L#2;
   Rear.Hook[2].HookOver := L#5560;
   Rear.Hook[2].HookUnderOffset := L#115;
   Rear.Hook[2].TelPos_1.TelPos := L#2;
   Rear.Hook[3].HookOver := L#4415;
   Rear.Hook[3].HookUnderOffset := L#115;
   Rear.Hook[3].TelPos_1.TelPos := L#2;
   Rear.Hook[4].HookOver := L#3260;
   Rear.Hook[4].HookUnderOffset := L#115;
   Rear.Hook[4].TelPos_1.TelPos := L#2;
   Rear.Hook[5].HookOver := L#2115;
   Rear.Hook[5].HookUnderOffset := L#115;
   Rear.Hook[5].TelPos_1.TelPos := L#2;
END_DATA_BLOCK

DATA_BLOCK "BR09_TR05"	// DB 293
VERSION : 0.1
  STRUCT
   Front : STRUCT
    Hook : ARRAY  [1 .. 10 ] OF UDT 102;
   END_STRUCT ;
   Rear : STRUCT
    Hook : ARRAY  [1 .. 10 ] OF UDT 102;
   END_STRUCT ;
  END_STRUCT ;	
BEGIN
   Front.Hook[1].HookOver := L#6703;
   Front.Hook[1].HookUnderOffset := L#115;
   Front.Hook[1].TelPos_1.TelPos := L#1;
   Front.Hook[2].HookOver := L#5560;
   Front.Hook[2].HookUnderOffset := L#115;
   Front.Hook[2].TelPos_1.TelPos := L#1;
   Front.Hook[3].HookOver := L#4415;
   Front.Hook[3].HookUnderOffset := L#115;
   Front.Hook[3].TelPos_1.TelPos := L#1;
   Front.Hook[4].HookOver := L#3260;
   Front.Hook[4].HookUnderOffset := L#115;
   Front.Hook[4].TelPos_1.TelPos := L#1;
   Front.Hook[5].HookOver := L#2115;
   Front.Hook[5].HookUnderOffset := L#115;
   Front.Hook[5].TelPos_1.TelPos := L#1;
   Rear.Hook[1].HookOver := L#6703;
   Rear.Hook[1].HookUnderOffset := L#115;
   Rear.Hook[1].TelPos_1.TelPos := L#2;
   Rear.Hook[2].HookOver := L#5560;
   Rear.Hook[2].HookUnderOffset := L#115;
   Rear.Hook[2].TelPos_1.TelPos := L#2;
   Rear.Hook[3].HookOver := L#4415;
   Rear.Hook[3].HookUnderOffset := L#115;
   Rear.Hook[3].TelPos_1.TelPos := L#2;
   Rear.Hook[4].HookOver := L#3260;
   Rear.Hook[4].HookUnderOffset := L#115;
   Rear.Hook[4].TelPos_1.TelPos := L#2;
   Rear.Hook[5].HookOver := L#2115;
   Rear.Hook[5].HookUnderOffset := L#115;
   Rear.Hook[5].TelPos_1.TelPos := L#2;
END_DATA_BLOCK

DATA_BLOCK "BR09_TR06"	// DB 294
VERSION : 0.1
  STRUCT
   Front : STRUCT
    Hook : ARRAY  [1 .. 10 ] OF UDT 102;
   END_STRUCT ;
   Rear : STRUCT
    Hook : ARRAY  [1 .. 10 ] OF UDT 102;
   END_STRUCT ;
  END_STRUCT ;	
BEGIN
   Front.Hook[1].HookOver := L#6703;
   Front.Hook[1].HookUnderOffset := L#115;
   Front.Hook[1].TelPos_1.TelPos := L#1;
   Front.Hook[2].HookOver := L#5560;
   Front.Hook[2].HookUnderOffset := L#115;
   Front.Hook[2].TelPos_1.TelPos := L#1;
   Front.Hook[3].HookOver := L#4415;
   Front.Hook[3].HookUnderOffset := L#115;
   Front.Hook[3].TelPos_1.TelPos := L#1;
   Front.Hook[4].HookOver := L#3260;
   Front.Hook[4].HookUnderOffset := L#115;
   Front.Hook[4].TelPos_1.TelPos := L#1;
   Front.Hook[5].HookOver := L#2115;
   Front.Hook[5].HookUnderOffset := L#115;
   Front.Hook[5].TelPos_1.TelPos := L#1;
   Rear.Hook[1].HookOver := L#6703;
   Rear.Hook[1].HookUnderOffset := L#115;
   Rear.Hook[1].TelPos_1.TelPos := L#2;
   Rear.Hook[2].HookOver := L#5560;
   Rear.Hook[2].HookUnderOffset := L#115;
   Rear.Hook[2].TelPos_1.TelPos := L#2;
   Rear.Hook[3].HookOver := L#4415;
   Rear.Hook[3].HookUnderOffset := L#115;
   Rear.Hook[3].TelPos_1.TelPos := L#2;
   Rear.Hook[4].HookOver := L#3260;
   Rear.Hook[4].HookUnderOffset := L#115;
   Rear.Hook[4].TelPos_1.TelPos := L#2;
   Rear.Hook[5].HookOver := L#2115;
   Rear.Hook[5].HookUnderOffset := L#115;
   Rear.Hook[5].TelPos_1.TelPos := L#2;
END_DATA_BLOCK

DATA_BLOCK "BR09_TR07"	// DB 295
VERSION : 0.1
  STRUCT
   Front : STRUCT
    Hook : ARRAY  [1 .. 10 ] OF UDT 102;
   END_STRUCT ;
   Rear : STRUCT
    Hook : ARRAY  [1 .. 10 ] OF UDT 102;
   END_STRUCT ;
  END_STRUCT ;	
BEGIN
   Front.Hook[1].HookOver := L#6703;
   Front.Hook[1].HookUnderOffset := L#115;
   Front.Hook[1].TelPos_1.TelPos := L#1;
   Front.Hook[2].HookOver := L#5560;
   Front.Hook[2].HookUnderOffset := L#115;
   Front.Hook[2].TelPos_1.TelPos := L#1;
   Front.Hook[3].HookOver := L#4415;
   Front.Hook[3].HookUnderOffset := L#115;
   Front.Hook[3].TelPos_1.TelPos := L#1;
   Front.Hook[4].HookOver := L#3260;
   Front.Hook[4].HookUnderOffset := L#115;
   Front.Hook[4].TelPos_1.TelPos := L#1;
   Front.Hook[5].HookOver := L#2115;
   Front.Hook[5].HookUnderOffset := L#115;
   Front.Hook[5].TelPos_1.TelPos := L#1;
   Rear.Hook[1].HookOver := L#6703;
   Rear.Hook[1].HookUnderOffset := L#115;
   Rear.Hook[1].TelPos_1.TelPos := L#2;
   Rear.Hook[2].HookOver := L#5560;
   Rear.Hook[2].HookUnderOffset := L#115;
   Rear.Hook[2].TelPos_1.TelPos := L#2;
   Rear.Hook[3].HookOver := L#4415;
   Rear.Hook[3].HookUnderOffset := L#115;
   Rear.Hook[3].TelPos_1.TelPos := L#2;
   Rear.Hook[4].HookOver := L#3260;
   Rear.Hook[4].HookUnderOffset := L#115;
   Rear.Hook[4].TelPos_1.TelPos := L#2;
   Rear.Hook[5].HookOver := L#2115;
   Rear.Hook[5].HookUnderOffset := L#115;
   Rear.Hook[5].TelPos_1.TelPos := L#2;
END_DATA_BLOCK

DATA_BLOCK "BR09_TR08"	// DB 296
VERSION : 0.1
  STRUCT
   Front : STRUCT
    Hook : ARRAY  [1 .. 10 ] OF UDT 102;
   END_STRUCT ;
   Rear : STRUCT
    Hook : ARRAY  [1 .. 10 ] OF UDT 102;
   END_STRUCT ;
  END_STRUCT ;	
BEGIN
   Front.Hook[1].HookOver := L#6703;
   Front.Hook[1].HookUnderOffset := L#115;
   Front.Hook[1].TelPos_1.TelPos := L#1;
   Front.Hook[2].HookOver := L#5560;
   Front.Hook[2].HookUnderOffset := L#115;
   Front.Hook[2].TelPos_1.TelPos := L#1;
   Front.Hook[3].HookOver := L#4415;
   Front.Hook[3].HookUnderOffset := L#115;
   Front.Hook[3].TelPos_1.TelPos := L#1;
   Front.Hook[4].HookOver := L#3260;
   Front.Hook[4].HookUnderOffset := L#115;
   Front.Hook[4].TelPos_1.TelPos := L#1;
   Front.Hook[5].HookOver := L#2115;
   Front.Hook[5].HookUnderOffset := L#115;
   Front.Hook[5].TelPos_1.TelPos := L#1;
   Rear.Hook[1].HookOver := L#6703;
   Rear.Hook[1].HookUnderOffset := L#115;
   Rear.Hook[1].TelPos_1.TelPos := L#2;
   Rear.Hook[2].HookOver := L#5560;
   Rear.Hook[2].HookUnderOffset := L#115;
   Rear.Hook[2].TelPos_1.TelPos := L#2;
   Rear.Hook[3].HookOver := L#4415;
   Rear.Hook[3].HookUnderOffset := L#115;
   Rear.Hook[3].TelPos_1.TelPos := L#2;
   Rear.Hook[4].HookOver := L#3260;
   Rear.Hook[4].HookUnderOffset := L#115;
   Rear.Hook[4].TelPos_1.TelPos := L#2;
   Rear.Hook[5].HookOver := L#2115;
   Rear.Hook[5].HookUnderOffset := L#115;
   Rear.Hook[5].TelPos_1.TelPos := L#2;
END_DATA_BLOCK

DATA_BLOCK "BR09_TR09"	// DB 297
VERSION : 0.1
  STRUCT
   Front : STRUCT
    Hook : ARRAY  [1 .. 10 ] OF UDT 102;
   END_STRUCT ;
   Rear : STRUCT
    Hook : ARRAY  [1 .. 10 ] OF UDT 102;
   END_STRUCT ;
  END_STRUCT ;	
BEGIN
END_DATA_BLOCK

DATA_BLOCK "BR09_TR10"	// DB 298
VERSION : 0.1
  STRUCT
   Front : STRUCT
    Hook : ARRAY  [1 .. 10 ] OF UDT 102;
   END_STRUCT ;
   Rear : STRUCT
    Hook : ARRAY  [1 .. 10 ] OF UDT 102;
   END_STRUCT ;
  END_STRUCT ;	
BEGIN
   Front.Hook[1].HookOver := L#6703;
   Front.Hook[1].HookUnderOffset := L#115;
   Front.Hook[2].HookOver := L#5560;
   Front.Hook[2].HookUnderOffset := L#115;
   Front.Hook[3].HookOver := L#4415;
   Front.Hook[3].HookUnderOffset := L#115;
   Front.Hook[3].TelPos_1.TelPos := L#1;
   Front.Hook[4].HookOver := L#3260;
   Front.Hook[4].HookUnderOffset := L#115;
   Front.Hook[4].TelPos_1.TelPos := L#1;
   Rear.Hook[1].HookOver := L#6703;
   Rear.Hook[1].HookUnderOffset := L#115;
   Rear.Hook[1].TelPos_1.TelPos := L#2;
   Rear.Hook[2].HookOver := L#5560;
   Rear.Hook[2].HookUnderOffset := L#115;
   Rear.Hook[2].TelPos_1.TelPos := L#2;
   Rear.Hook[3].HookOver := L#4415;
   Rear.Hook[3].HookUnderOffset := L#115;
   Rear.Hook[3].TelPos_1.TelPos := L#2;
   Rear.Hook[4].HookOver := L#3260;
   Rear.Hook[4].HookUnderOffset := L#115;
   Rear.Hook[4].TelPos_1.TelPos := L#2;
END_DATA_BLOCK

DATA_BLOCK "BR09_TR11"	// DB 299
VERSION : 0.1
  STRUCT
   Front : STRUCT
    Hook : ARRAY  [1 .. 10 ] OF UDT 102;
   END_STRUCT ;
   Rear : STRUCT
    Hook : ARRAY  [1 .. 10 ] OF UDT 102;
   END_STRUCT ;
  END_STRUCT ;	
BEGIN
END_DATA_BLOCK

DATA_BLOCK "BR10_TR01"	// DB 300
VERSION : 0.1
  STRUCT
   Front : STRUCT
    Hook : ARRAY  [1 .. 10 ] OF UDT 102;
   END_STRUCT ;
   Rear : STRUCT
    Hook : ARRAY  [1 .. 10 ] OF UDT 102;
   END_STRUCT ;
  END_STRUCT ;	
BEGIN
   Front.Hook[1].HookOver := L#6716;
   Front.Hook[1].HookUnderOffset := L#115;
   Front.Hook[1].TelPos_1.TelPos := L#1;
   Front.Hook[2].HookOver := L#5566;
   Front.Hook[2].HookUnderOffset := L#115;
   Front.Hook[2].TelPos_1.TelPos := L#1;
   Front.Hook[3].HookOver := L#4416;
   Front.Hook[3].HookUnderOffset := L#115;
   Front.Hook[3].TelPos_1.TelPos := L#1;
   Front.Hook[4].HookOver := L#3266;
   Front.Hook[4].HookUnderOffset := L#115;
   Front.Hook[4].TelPos_1.TelPos := L#1;
   Rear.Hook[1].HookOver := L#6716;
   Rear.Hook[1].HookUnderOffset := L#115;
   Rear.Hook[1].TelPos_1.TelPos := L#2;
   Rear.Hook[2].HookOver := L#5566;
   Rear.Hook[2].HookUnderOffset := L#115;
   Rear.Hook[2].TelPos_1.TelPos := L#2;
   Rear.Hook[3].HookOver := L#4416;
   Rear.Hook[3].HookUnderOffset := L#115;
   Rear.Hook[3].TelPos_1.TelPos := L#2;
   Rear.Hook[4].HookOver := L#3266;
   Rear.Hook[4].HookUnderOffset := L#115;
   Rear.Hook[4].TelPos_1.TelPos := L#2;
END_DATA_BLOCK

DATA_BLOCK "BR10_TR02"	// DB 301
VERSION : 0.1
  STRUCT
   Front : STRUCT
    Hook : ARRAY  [1 .. 10 ] OF UDT 102;
   END_STRUCT ;
   Rear : STRUCT
    Hook : ARRAY  [1 .. 10 ] OF UDT 102;
   END_STRUCT ;
  END_STRUCT ;	
BEGIN
   Front.Hook[1].HookOver := L#6703;
   Front.Hook[1].HookUnderOffset := L#115;
   Front.Hook[1].TelPos_1.TelPos := L#1;
   Front.Hook[2].HookOver := L#5560;
   Front.Hook[2].HookUnderOffset := L#115;
   Front.Hook[2].TelPos_1.TelPos := L#1;
   Front.Hook[3].HookOver := L#4415;
   Front.Hook[3].HookUnderOffset := L#115;
   Front.Hook[3].TelPos_1.TelPos := L#1;
   Front.Hook[4].HookOver := L#3260;
   Front.Hook[4].HookUnderOffset := L#115;
   Front.Hook[4].TelPos_1.TelPos := L#1;
   Front.Hook[5].HookOver := L#2115;
   Front.Hook[5].HookUnderOffset := L#115;
   Front.Hook[5].TelPos_1.TelPos := L#1;
   Rear.Hook[1].HookOver := L#6703;
   Rear.Hook[1].HookUnderOffset := L#115;
   Rear.Hook[1].TelPos_1.TelPos := L#2;
   Rear.Hook[2].HookOver := L#5560;
   Rear.Hook[2].HookUnderOffset := L#115;
   Rear.Hook[2].TelPos_1.TelPos := L#2;
   Rear.Hook[3].HookOver := L#4415;
   Rear.Hook[3].HookUnderOffset := L#115;
   Rear.Hook[3].TelPos_1.TelPos := L#2;
   Rear.Hook[4].HookOver := L#3260;
   Rear.Hook[4].HookUnderOffset := L#115;
   Rear.Hook[4].TelPos_1.TelPos := L#2;
   Rear.Hook[5].HookOver := L#2115;
   Rear.Hook[5].HookUnderOffset := L#115;
   Rear.Hook[5].TelPos_1.TelPos := L#2;
END_DATA_BLOCK

DATA_BLOCK "BR10_TR03"	// DB 302
VERSION : 0.1
  STRUCT
   Front : STRUCT
    Hook : ARRAY  [1 .. 10 ] OF UDT 102;
   END_STRUCT ;
   Rear : STRUCT
    Hook : ARRAY  [1 .. 10 ] OF UDT 102;
   END_STRUCT ;
  END_STRUCT ;	
BEGIN
   Front.Hook[1].HookOver := L#6703;
   Front.Hook[1].HookUnderOffset := L#115;
   Front.Hook[1].TelPos_1.TelPos := L#1;
   Front.Hook[2].HookOver := L#5560;
   Front.Hook[2].HookUnderOffset := L#115;
   Front.Hook[2].TelPos_1.TelPos := L#1;
   Front.Hook[3].HookOver := L#4415;
   Front.Hook[3].HookUnderOffset := L#115;
   Front.Hook[3].TelPos_1.TelPos := L#1;
   Front.Hook[4].HookOver := L#3260;
   Front.Hook[4].HookUnderOffset := L#115;
   Front.Hook[4].TelPos_1.TelPos := L#1;
   Front.Hook[5].HookOver := L#2115;
   Front.Hook[5].HookUnderOffset := L#115;
   Front.Hook[5].TelPos_1.TelPos := L#1;
   Rear.Hook[1].HookOver := L#6703;
   Rear.Hook[1].HookUnderOffset := L#115;
   Rear.Hook[1].TelPos_1.TelPos := L#2;
   Rear.Hook[2].HookOver := L#5560;
   Rear.Hook[2].HookUnderOffset := L#115;
   Rear.Hook[2].TelPos_1.TelPos := L#2;
   Rear.Hook[3].HookOver := L#4415;
   Rear.Hook[3].HookUnderOffset := L#115;
   Rear.Hook[3].TelPos_1.TelPos := L#2;
   Rear.Hook[4].HookOver := L#3260;
   Rear.Hook[4].HookUnderOffset := L#115;
   Rear.Hook[4].TelPos_1.TelPos := L#2;
   Rear.Hook[5].HookOver := L#2115;
   Rear.Hook[5].HookUnderOffset := L#115;
   Rear.Hook[5].TelPos_1.TelPos := L#2;
END_DATA_BLOCK

DATA_BLOCK "BR10_TR04"	// DB 303
VERSION : 0.1
  STRUCT
   Front : STRUCT
    Hook : ARRAY  [1 .. 10 ] OF UDT 102;
   END_STRUCT ;
   Rear : STRUCT
    Hook : ARRAY  [1 .. 10 ] OF UDT 102;
   END_STRUCT ;
  END_STRUCT ;	
BEGIN
   Front.Hook[1].HookOver := L#6703;
   Front.Hook[1].HookUnderOffset := L#115;
   Front.Hook[1].TelPos_1.TelPos := L#1;
   Front.Hook[2].HookOver := L#5560;
   Front.Hook[2].HookUnderOffset := L#115;
   Front.Hook[2].TelPos_1.TelPos := L#1;
   Front.Hook[3].HookOver := L#4415;
   Front.Hook[3].HookUnderOffset := L#115;
   Front.Hook[3].TelPos_1.TelPos := L#1;
   Front.Hook[4].HookOver := L#3260;
   Front.Hook[4].HookUnderOffset := L#115;
   Front.Hook[4].TelPos_1.TelPos := L#1;
   Front.Hook[5].HookOver := L#2115;
   Front.Hook[5].HookUnderOffset := L#115;
   Front.Hook[5].TelPos_1.TelPos := L#1;
   Rear.Hook[1].HookOver := L#6703;
   Rear.Hook[1].HookUnderOffset := L#115;
   Rear.Hook[1].TelPos_1.TelPos := L#2;
   Rear.Hook[2].HookOver := L#5560;
   Rear.Hook[2].HookUnderOffset := L#115;
   Rear.Hook[2].TelPos_1.TelPos := L#2;
   Rear.Hook[3].HookOver := L#4415;
   Rear.Hook[3].HookUnderOffset := L#115;
   Rear.Hook[3].TelPos_1.TelPos := L#2;
   Rear.Hook[4].HookOver := L#3260;
   Rear.Hook[4].HookUnderOffset := L#115;
   Rear.Hook[4].TelPos_1.TelPos := L#2;
   Rear.Hook[5].HookOver := L#2115;
   Rear.Hook[5].HookUnderOffset := L#115;
   Rear.Hook[5].TelPos_1.TelPos := L#2;
END_DATA_BLOCK

DATA_BLOCK "BR10_TR05"	// DB 304
VERSION : 0.1
  STRUCT
   Front : STRUCT
    Hook : ARRAY  [1 .. 10 ] OF UDT 102;
   END_STRUCT ;
   Rear : STRUCT
    Hook : ARRAY  [1 .. 10 ] OF UDT 102;
   END_STRUCT ;
  END_STRUCT ;	
BEGIN
   Front.Hook[1].HookOver := L#6703;
   Front.Hook[1].HookUnderOffset := L#115;
   Front.Hook[1].TelPos_1.TelPos := L#1;
   Front.Hook[2].HookOver := L#5560;
   Front.Hook[2].HookUnderOffset := L#115;
   Front.Hook[2].TelPos_1.TelPos := L#1;
   Front.Hook[3].HookOver := L#4415;
   Front.Hook[3].HookUnderOffset := L#115;
   Front.Hook[3].TelPos_1.TelPos := L#1;
   Front.Hook[4].HookOver := L#3260;
   Front.Hook[4].HookUnderOffset := L#115;
   Front.Hook[4].TelPos_1.TelPos := L#1;
   Front.Hook[5].HookOver := L#2115;
   Front.Hook[5].HookUnderOffset := L#115;
   Front.Hook[5].TelPos_1.TelPos := L#1;
   Rear.Hook[1].HookOver := L#6703;
   Rear.Hook[1].HookUnderOffset := L#115;
   Rear.Hook[1].TelPos_1.TelPos := L#2;
   Rear.Hook[2].HookOver := L#5560;
   Rear.Hook[2].HookUnderOffset := L#115;
   Rear.Hook[2].TelPos_1.TelPos := L#2;
   Rear.Hook[3].HookOver := L#4415;
   Rear.Hook[3].HookUnderOffset := L#115;
   Rear.Hook[3].TelPos_1.TelPos := L#2;
   Rear.Hook[4].HookOver := L#3260;
   Rear.Hook[4].HookUnderOffset := L#115;
   Rear.Hook[4].TelPos_1.TelPos := L#2;
   Rear.Hook[5].HookOver := L#2115;
   Rear.Hook[5].HookUnderOffset := L#115;
   Rear.Hook[5].TelPos_1.TelPos := L#2;
END_DATA_BLOCK

DATA_BLOCK "BR10_TR06"	// DB 305
VERSION : 0.1
  STRUCT
   Front : STRUCT
    Hook : ARRAY  [1 .. 10 ] OF UDT 102;
   END_STRUCT ;
   Rear : STRUCT
    Hook : ARRAY  [1 .. 10 ] OF UDT 102;
   END_STRUCT ;
  END_STRUCT ;	
BEGIN
   Front.Hook[1].HookOver := L#6703;
   Front.Hook[1].HookUnderOffset := L#115;
   Front.Hook[1].TelPos_1.TelPos := L#1;
   Front.Hook[2].HookOver := L#5560;
   Front.Hook[2].HookUnderOffset := L#115;
   Front.Hook[2].TelPos_1.TelPos := L#1;
   Front.Hook[3].HookOver := L#4415;
   Front.Hook[3].HookUnderOffset := L#115;
   Front.Hook[3].TelPos_1.TelPos := L#1;
   Front.Hook[4].HookOver := L#3260;
   Front.Hook[4].HookUnderOffset := L#115;
   Front.Hook[4].TelPos_1.TelPos := L#1;
   Front.Hook[5].HookOver := L#2115;
   Front.Hook[5].HookUnderOffset := L#115;
   Front.Hook[5].TelPos_1.TelPos := L#1;
   Rear.Hook[1].HookOver := L#6703;
   Rear.Hook[1].HookUnderOffset := L#115;
   Rear.Hook[1].TelPos_1.TelPos := L#2;
   Rear.Hook[2].HookOver := L#5560;
   Rear.Hook[2].HookUnderOffset := L#115;
   Rear.Hook[2].TelPos_1.TelPos := L#2;
   Rear.Hook[3].HookOver := L#4415;
   Rear.Hook[3].HookUnderOffset := L#115;
   Rear.Hook[3].TelPos_1.TelPos := L#2;
   Rear.Hook[4].HookOver := L#3260;
   Rear.Hook[4].HookUnderOffset := L#115;
   Rear.Hook[4].TelPos_1.TelPos := L#2;
   Rear.Hook[5].HookOver := L#2115;
   Rear.Hook[5].HookUnderOffset := L#115;
   Rear.Hook[5].TelPos_1.TelPos := L#2;
END_DATA_BLOCK

DATA_BLOCK "BR10_TR07"	// DB 306
VERSION : 0.1
  STRUCT
   Front : STRUCT
    Hook : ARRAY  [1 .. 10 ] OF UDT 102;
   END_STRUCT ;
   Rear : STRUCT
    Hook : ARRAY  [1 .. 10 ] OF UDT 102;
   END_STRUCT ;
  END_STRUCT ;	
BEGIN
   Front.Hook[1].HookOver := L#6703;
   Front.Hook[1].HookUnderOffset := L#115;
   Front.Hook[1].TelPos_1.TelPos := L#1;
   Front.Hook[2].HookOver := L#5560;
   Front.Hook[2].HookUnderOffset := L#115;
   Front.Hook[2].TelPos_1.TelPos := L#1;
   Front.Hook[3].HookOver := L#4415;
   Front.Hook[3].HookUnderOffset := L#115;
   Front.Hook[3].TelPos_1.TelPos := L#1;
   Front.Hook[4].HookOver := L#3260;
   Front.Hook[4].HookUnderOffset := L#115;
   Front.Hook[4].TelPos_1.TelPos := L#1;
   Front.Hook[5].HookOver := L#2115;
   Front.Hook[5].HookUnderOffset := L#115;
   Front.Hook[5].TelPos_1.TelPos := L#1;
   Rear.Hook[1].HookOver := L#6703;
   Rear.Hook[1].HookUnderOffset := L#115;
   Rear.Hook[1].TelPos_1.TelPos := L#2;
   Rear.Hook[2].HookOver := L#5560;
   Rear.Hook[2].HookUnderOffset := L#115;
   Rear.Hook[2].TelPos_1.TelPos := L#2;
   Rear.Hook[3].HookOver := L#4415;
   Rear.Hook[3].HookUnderOffset := L#115;
   Rear.Hook[3].TelPos_1.TelPos := L#2;
   Rear.Hook[4].HookOver := L#3260;
   Rear.Hook[4].HookUnderOffset := L#115;
   Rear.Hook[4].TelPos_1.TelPos := L#2;
   Rear.Hook[5].HookOver := L#2115;
   Rear.Hook[5].HookUnderOffset := L#115;
   Rear.Hook[5].TelPos_1.TelPos := L#2;
END_DATA_BLOCK

DATA_BLOCK "BR10_TR08"	// DB 307
VERSION : 0.1
  STRUCT
   Front : STRUCT
    Hook : ARRAY  [1 .. 10 ] OF UDT 102;
   END_STRUCT ;
   Rear : STRUCT
    Hook : ARRAY  [1 .. 10 ] OF UDT 102;
   END_STRUCT ;
  END_STRUCT ;	
BEGIN
   Front.Hook[1].HookOver := L#6703;
   Front.Hook[1].HookUnderOffset := L#115;
   Front.Hook[1].TelPos_1.TelPos := L#1;
   Front.Hook[2].HookOver := L#5560;
   Front.Hook[2].HookUnderOffset := L#115;
   Front.Hook[2].TelPos_1.TelPos := L#1;
   Front.Hook[3].HookOver := L#4415;
   Front.Hook[3].HookUnderOffset := L#115;
   Front.Hook[3].TelPos_1.TelPos := L#1;
   Front.Hook[4].HookOver := L#3260;
   Front.Hook[4].HookUnderOffset := L#115;
   Front.Hook[4].TelPos_1.TelPos := L#1;
   Front.Hook[5].HookOver := L#2115;
   Front.Hook[5].HookUnderOffset := L#115;
   Front.Hook[5].TelPos_1.TelPos := L#1;
   Rear.Hook[1].HookOver := L#6703;
   Rear.Hook[1].HookUnderOffset := L#115;
   Rear.Hook[1].TelPos_1.TelPos := L#2;
   Rear.Hook[2].HookOver := L#5560;
   Rear.Hook[2].HookUnderOffset := L#115;
   Rear.Hook[2].TelPos_1.TelPos := L#2;
   Rear.Hook[3].HookOver := L#4415;
   Rear.Hook[3].HookUnderOffset := L#115;
   Rear.Hook[3].TelPos_1.TelPos := L#2;
   Rear.Hook[4].HookOver := L#3260;
   Rear.Hook[4].HookUnderOffset := L#115;
   Rear.Hook[4].TelPos_1.TelPos := L#2;
   Rear.Hook[5].HookOver := L#2115;
   Rear.Hook[5].HookUnderOffset := L#115;
   Rear.Hook[5].TelPos_1.TelPos := L#2;
END_DATA_BLOCK

DATA_BLOCK "BR10_TR09"	// DB 308
VERSION : 0.1
  STRUCT
   Front : STRUCT
    Hook : ARRAY  [1 .. 10 ] OF UDT 102;
   END_STRUCT ;
   Rear : STRUCT
    Hook : ARRAY  [1 .. 10 ] OF UDT 102;
   END_STRUCT ;
  END_STRUCT ;	
BEGIN
END_DATA_BLOCK

DATA_BLOCK "BR10_TR10"	// DB 309
VERSION : 0.1
  STRUCT
   Front : STRUCT
    Hook : ARRAY  [1 .. 10 ] OF UDT 102;
   END_STRUCT ;
   Rear : STRUCT
    Hook : ARRAY  [1 .. 10 ] OF UDT 102;
   END_STRUCT ;
  END_STRUCT ;	
BEGIN
   Front.Hook[1].HookOver := L#6703;
   Front.Hook[1].HookUnderOffset := L#115;
   Front.Hook[2].HookOver := L#5560;
   Front.Hook[2].HookUnderOffset := L#115;
   Front.Hook[3].HookOver := L#4415;
   Front.Hook[3].HookUnderOffset := L#115;
   Front.Hook[3].TelPos_1.TelPos := L#1;
   Front.Hook[4].HookOver := L#3260;
   Front.Hook[4].HookUnderOffset := L#115;
   Front.Hook[4].TelPos_1.TelPos := L#1;
   Rear.Hook[1].HookOver := L#6703;
   Rear.Hook[1].HookUnderOffset := L#115;
   Rear.Hook[1].TelPos_1.TelPos := L#2;
   Rear.Hook[2].HookOver := L#5560;
   Rear.Hook[2].HookUnderOffset := L#115;
   Rear.Hook[2].TelPos_1.TelPos := L#2;
   Rear.Hook[3].HookOver := L#4415;
   Rear.Hook[3].HookUnderOffset := L#115;
   Rear.Hook[3].TelPos_1.TelPos := L#2;
   Rear.Hook[4].HookOver := L#3260;
   Rear.Hook[4].HookUnderOffset := L#115;
   Rear.Hook[4].TelPos_1.TelPos := L#2;
END_DATA_BLOCK

DATA_BLOCK "BR10_TR11"	// DB 310
VERSION : 0.1
  STRUCT
   Front : STRUCT
    Hook : ARRAY  [1 .. 10 ] OF UDT 102;
   END_STRUCT ;
   Rear : STRUCT
    Hook : ARRAY  [1 .. 10 ] OF UDT 102;
   END_STRUCT ;
  END_STRUCT ;	
BEGIN
END_DATA_BLOCK

DATA_BLOCK "BR11_TR01"	// DB 311
VERSION : 0.1
  STRUCT
   Front : STRUCT
    Hook : ARRAY  [1 .. 10 ] OF UDT 102;
   END_STRUCT ;
   Rear : STRUCT
    Hook : ARRAY  [1 .. 10 ] OF UDT 102;
   END_STRUCT ;
  END_STRUCT ;	
BEGIN
   Front.Hook[1].HookOver := L#2000;
   Front.Hook[1].HookUnderOffset := L#115;
   Front.Hook[1].TelPos_1.TelPos := L#1;
   Rear.Hook[1].HookOver := L#2000;
   Rear.Hook[1].HookUnderOffset := L#115;
   Rear.Hook[1].TelPos_1.TelPos := L#2;
END_DATA_BLOCK

DATA_BLOCK "BR11_TR02"	// DB 312
VERSION : 0.1
  STRUCT
   Front : STRUCT
    Hook : ARRAY  [1 .. 10 ] OF UDT 102;
   END_STRUCT ;
   Rear : STRUCT
    Hook : ARRAY  [1 .. 10 ] OF UDT 102;
   END_STRUCT ;
  END_STRUCT ;	
BEGIN
   Front.Hook[1].HookOver := L#2000;
   Front.Hook[1].HookUnderOffset := L#115;
   Front.Hook[1].TelPos_1.TelPos := L#1;
   Rear.Hook[1].HookOver := L#2000;
   Rear.Hook[1].HookUnderOffset := L#115;
   Rear.Hook[1].TelPos_1.TelPos := L#2;
END_DATA_BLOCK

DATA_BLOCK "LIF_Pos"	// DB 350
VERSION : 0.1
  STRUCT
   Front : STRUCT
    Hook : ARRAY  [1 .. 10 ] OF UDT 102;
   END_STRUCT ;
   Rear : STRUCT
    Hook : ARRAY  [1 .. 10 ] OF UDT 102;
   END_STRUCT ;
  END_STRUCT ;	
BEGIN
END_DATA_BLOCK

DATA_BLOCK "ProfiNet"	// DB 400
VERSION : 0.0
  STRUCT
   STAT0 : ARRAY  [-32768 .. -31295 ] OF BYTE ;
  END_STRUCT ;	
BEGIN
   STAT0[-32685] := B#16#1;
   STAT0[-32683] := B#16#1;
   STAT0[-32681] := B#16#1;
   STAT0[-32679] := B#16#1;
   STAT0[-31744] := B#16#90;
   STAT0[-31743] := B#16#1;
   STAT0[-31742] := B#16#1;
   STAT0[-31737] := B#16#2;
END_DATA_BLOCK

